KUKA KRL program: f1_Kuka_APT222T02S22.SRC

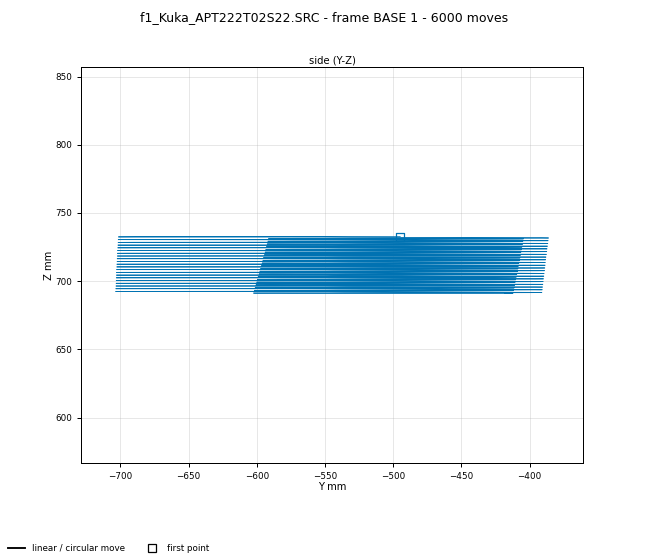
[picture p0: tool path of f1_Kuka_APT222T02S22.SRC in frame BASE 1, 6000 of 6001 moves have a stored position in this frame; points joined in program order, loops and branches not executed]
&ACCESS RVP
&REL 2
&PARAM TEMPLATE = C:\KRC\Roboter\Template\vorgabe
&PARAM EDITMASK = *
DEF f1_Kuka_APT222T02S22()


;FOLD INI;%{PE}%V3.2.0,%MKUKATPBASIS,%CINIT,%VCOMMON,%P
  ;FOLD BAS INI;%{E}%V3.2.0,%MKUKATPBASIS,%CINIT,%VINIT,%P
    GLOBAL INTERRUPT DECL 3 WHEN $STOPMESS==TRUE DO IR_STOPM ( )
    INTERRUPT ON 3
    BAS (#INITMOV,0 )
  ;ENDFOLD (BAS INI)
  ;FOLD USER INI;%{E}%V3.2.0,%MKUKATPUSER,%CINIT,%VINIT,%P
    ;Make your modifications here
  ;ENDFOLD (USER INI)
;ENDFOLD (INI)


;*** Make Null PTP Move
  PTP $pos_act

;*** Auto Load The Correct TOOL Data
  $tool=tool_data[2]

;*** Auto Load The Correct BASE Data
  $base=base_data[1]

  $ADVANCE = 5

;*** Restate Last Velocity
MMPM(30000.0)
SetRPM(8000)
LIN {X -0.072,Y -494.811,Z 732.685,A 0.000,B 0.000,C 90.000,E1 339.263} C_DIS
LIN {X 0.062,Y -499.458,Z 732.683,A 0.000,B 0.000,C 90.000,E1 338.847} C_DIS
LIN {X -0.040,Y -508.556,Z 732.679,A 0.000,B 0.000,C 90.000,E1 338.230} C_DIS
LIN {X -0.102,Y -530.986,Z 732.671,A 0.000,B 0.000,C 90.000,E1 336.847} C_DIS
LIN {X -0.056,Y -538.848,Z 732.669,A 0.000,B 0.000,C 90.000,E1 336.357} C_DIS
LIN {X 0.219,Y -546.203,Z 732.666,A 0.000,B 0.000,C 90.000,E1 335.793} C_DIS
LIN {X -0.007,Y -551.872,Z 732.663,A 0.000,B 0.000,C 90.000,E1 335.357} C_DIS
LIN {X 0.256,Y -559.941,Z 732.659,A 0.000,B 0.000,C 90.000,E1 334.588} C_DIS
LIN {X -0.047,Y -566.520,Z 732.655,A 0.000,B 0.000,C 90.000,E1 333.973} C_DIS
LIN {X -0.138,Y -575.282,Z 732.650,A 0.000,B 0.000,C 90.000,E1 333.050} C_DIS
LIN {X -0.034,Y -582.251,Z 732.646,A 0.000,B 0.000,C 90.000,E1 332.231} C_DIS
LIN {X -0.259,Y -591.121,Z 732.640,A 0.000,B 0.000,C 90.000,E1 331.179} C_DIS
LIN {X 0.245,Y -597.384,Z 732.635,A 0.000,B 0.000,C 90.000,E1 330.333} C_DIS
LIN {X 0.263,Y -604.345,Z 732.630,A 0.000,B 0.000,C 90.000,E1 329.410} C_DIS
LIN {X -0.134,Y -610.077,Z 732.626,A 0.000,B 0.000,C 90.000,E1 328.663} C_DIS
LIN {X 0.337,Y -617.212,Z 732.620,A 0.000,B 0.000,C 90.000,E1 327.582} C_DIS
LIN {X 0.048,Y -623.875,Z 732.614,A 0.000,B 0.000,C 90.000,E1 326.580} C_DIS
LIN {X 0.187,Y -628.508,Z 732.610,A 0.000,B 0.000,C 90.000,E1 325.801} C_DIS
LIN {X 0.019,Y -632.989,Z 732.606,A 0.000,B 0.000,C 90.000,E1 325.055} C_DIS
LIN {X -0.254,Y -637.926,Z 732.601,A 0.000,B 0.000,C 90.000,E1 324.196} C_DIS
LIN {X 0.036,Y -641.902,Z 732.597,A 0.000,B 0.000,C 90.000,E1 323.417} C_DIS
LIN {X -0.147,Y -645.788,Z 732.593,A 0.000,B 0.000,C 90.000,E1 322.683} C_DIS
LIN {X 0.221,Y -649.398,Z 732.589,A 0.000,B 0.000,C 90.000,E1 321.904} C_DIS
LIN {X 0.047,Y -653.994,Z 732.583,A 0.000,B 0.000,C 90.000,E1 320.928} C_DIS
LIN {X -0.062,Y -658.317,Z 732.578,A 0.000,B 0.000,C 90.000,E1 319.952} C_DIS
LIN {X 0.386,Y -662.353,Z 732.572,A 0.000,B 0.000,C 90.000,E1 318.933} C_DIS
LIN {X -0.109,Y -665.266,Z 732.568,A 0.000,B 0.000,C 90.000,E1 318.243} C_DIS
LIN {X 0.365,Y -667.979,Z 732.564,A 0.000,B 0.000,C 90.000,E1 317.472} C_DIS
LIN {X -0.061,Y -672.104,Z 732.557,A 0.000,B 0.000,C 90.000,E1 316.296} C_DIS
LIN {X 0.018,Y -675.195,Z 732.552,A 0.000,B 0.000,C 90.000,E1 315.324} C_DIS
LIN {X 0.141,Y -678.120,Z 732.547,A 0.000,B 0.000,C 90.000,E1 314.352} C_DIS
LIN {X -0.126,Y -681.503,Z 732.540,A 0.000,B 0.000,C 90.000,E1 313.176} C_DIS
LIN {X -0.340,Y -684.578,Z 732.533,A 0.000,B 0.000,C 90.000,E1 312.000} C_DIS
LIN {X 0.003,Y -687.418,Z 732.527,A 0.000,B 0.000,C 90.000,E1 310.782} C_DIS
LIN {X -0.202,Y -689.405,Z 732.521,A 0.000,B 0.000,C 90.000,E1 309.850} C_DIS
LIN {X -0.297,Y -691.088,Z 732.516,A 0.000,B 0.000,C 90.000,E1 308.910} C_DIS
LIN {X 0.064,Y -692.544,Z 732.511,A 0.000,B 0.000,C 90.000,E1 307.935} C_DIS
LIN {X 0.210,Y -694.120,Z 732.504,A 0.000,B 0.000,C 90.000,E1 306.744} C_DIS
LIN {X 0.181,Y -695.226,Z 732.499,A 0.000,B 0.000,C 90.000,E1 305.804} C_DIS
LIN {X -0.244,Y -696.182,Z 732.494,A 0.000,B 0.000,C 90.000,E1 304.898} C_DIS
LIN {X 0.204,Y -697.306,Z 732.486,A 0.000,B 0.000,C 90.000,E1 303.452} C_DIS
LIN {X -0.291,Y -698.505,Z 732.478,A 0.000,B 0.000,C 90.000,E1 302.084} C_DIS
LIN {X 0.163,Y -699.440,Z 732.472,A 0.000,B 0.000,C 90.000,E1 300.875} C_DIS
LIN {X 0.011,Y -699.898,Z 732.466,A 0.000,B 0.000,C 90.000,E1 299.951} C_DIS
LIN {X 0.137,Y -700.212,Z 732.460,A 0.000,B 0.000,C 90.000,E1 298.771} C_DIS
LIN {X -0.162,Y -700.761,Z 732.450,A 0.000,B 0.000,C 90.000,E1 296.924} C_DIS
LIN {X -0.116,Y -701.515,Z 732.440,A 0.000,B 0.000,C 90.000,E1 295.283} C_DIS
LIN {X -0.220,Y -701.426,Z 732.437,A 0.000,B 0.000,C 90.000,E1 294.591} C_DIS
LIN {X 0.329,Y -700.180,Z 732.434,A 0.000,B 0.000,C 90.000,E1 294.079} C_DIS
LIN {X -0.324,Y -699.415,Z 732.433,A 0.000,B 0.000,C 90.000,E1 293.898} C_DIS
LIN {X -0.190,Y -698.702,Z 732.432,A 0.000,B 0.000,C 90.000,E1 293.770} C_DIS
LIN {X 0.076,Y -696.517,Z 732.431,A 0.000,B 0.000,C 90.000,E1 293.515} C_DIS
LIN {X 0.347,Y -694.183,Z 732.429,A 0.000,B 0.000,C 90.000,E1 293.259} C_DIS
LIN {X 0.217,Y -692.875,Z 732.429,A 0.000,B 0.000,C 90.000,E1 293.153} C_DIS
LIN {X -0.223,Y -690.907,Z 732.428,A 0.000,B 0.000,C 90.000,E1 293.078} C_DIS
LIN {X -0.185,Y -686.403,Z 732.427,A 0.000,B 0.000,C 90.000,E1 292.898} C_DIS
LIN {X -0.121,Y -682.477,Z 732.427,A 0.000,B 0.000,C 90.000,E1 292.770} C_DIS
LIN {X 0.202,Y -676.428,Z 732.426,A 0.000,B 0.000,C 90.000,E1 292.589} C_DIS
LIN {X 0.149,Y -666.176,Z 732.425,A 0.000,B 0.000,C 90.000,E1 292.461} C_DIS
LIN {X 0.096,Y -652.560,Z 732.424,A 0.000,B 0.000,C 90.000,E1 292.280} C_DIS
LIN {X -0.358,Y -642.712,Z 732.423,A 0.000,B 0.000,C 90.000,E1 292.153} C_DIS
LIN {X 0.011,Y -629.339,Z 732.421,A 0.000,B 0.000,C 90.000,E1 291.844} C_DIS
LIN {X -0.078,Y -608.968,Z 732.419,A 0.000,B 0.000,C 90.000,E1 291.334} C_DIS
LIN {X -0.262,Y -581.079,Z 732.414,A 0.000,B 0.000,C 90.000,E1 290.556} C_DIS
LIN {X -0.251,Y -571.987,Z 732.413,A 0.000,B 0.000,C 90.000,E1 290.301} C_DIS
LIN {X 0.122,Y -566.747,Z 732.412,A 0.000,B 0.000,C 90.000,E1 290.120} C_DIS
LIN {X 0.007,Y -561.140,Z 732.411,A 0.000,B 0.000,C 90.000,E1 289.939} C_DIS
LIN {X -0.094,Y -556.625,Z 732.409,A 0.000,B 0.000,C 90.000,E1 289.685} C_DIS
LIN {X -0.122,Y -556.604,Z 732.409,A 0.000,B 0.000,C 90.000,E1 289.685} C_DIS
LIN {X -0.115,Y -555.581,Z 732.408,A 0.000,B 0.000,C 90.000,E1 289.504} C_DIS
LIN {X -0.129,Y -554.925,Z 732.406,A 0.000,B 0.000,C 90.000,E1 289.087} C_DIS
LIN {X 0.037,Y -554.116,Z 732.394,A 0.000,B 0.000,C 90.000,E1 286.913} C_DIS
LIN {X -0.146,Y -553.591,Z 732.386,A 0.000,B 0.000,C 90.000,E1 285.536} C_DIS
LIN {X -0.130,Y -552.835,Z 732.374,A 0.000,B 0.000,C 90.000,E1 283.300} C_DIS
LIN {X 0.286,Y -552.159,Z 732.363,A 0.000,B 0.000,C 90.000,E1 281.299} C_DIS
LIN {X 0.231,Y -551.598,Z 732.355,A 0.000,B 0.000,C 90.000,E1 279.905} C_DIS
LIN {X 0.170,Y -550.915,Z 732.347,A 0.000,B 0.000,C 90.000,E1 278.511} C_DIS
LIN {X 0.123,Y -550.135,Z 732.338,A 0.000,B 0.000,C 90.000,E1 276.834} C_DIS
LIN {X -0.008,Y -549.461,Z 732.329,A 0.000,B 0.000,C 90.000,E1 275.163} C_DIS
LIN {X 0.258,Y -549.002,Z 732.323,A 0.000,B 0.000,C 90.000,E1 274.012} C_DIS
LIN {X 0.072,Y -548.128,Z 732.312,A 0.000,B 0.000,C 90.000,E1 272.064} C_DIS
LIN {X -0.267,Y -547.557,Z 732.305,A 0.000,B 0.000,C 90.000,E1 270.974} C_DIS
LIN {X 0.009,Y -546.610,Z 732.296,A 0.000,B 0.000,C 90.000,E1 269.255} C_DIS
LIN {X 0.274,Y -545.503,Z 732.286,A 0.000,B 0.000,C 90.000,E1 267.535} C_DIS
LIN {X -0.068,Y -544.592,Z 732.279,A 0.000,B 0.000,C 90.000,E1 266.159} C_DIS
LIN {X 0.151,Y -543.656,Z 732.271,A 0.000,B 0.000,C 90.000,E1 264.723} C_DIS
LIN {X -0.122,Y -542.404,Z 732.261,A 0.000,B 0.000,C 90.000,E1 263.053} C_DIS
LIN {X 0.032,Y -541.731,Z 732.257,A 0.000,B 0.000,C 90.000,E1 262.186} C_DIS
LIN {X -0.058,Y -540.061,Z 732.246,A 0.000,B 0.000,C 90.000,E1 260.208} C_DIS
LIN {X -0.254,Y -538.600,Z 732.236,A 0.000,B 0.000,C 90.000,E1 258.522} C_DIS
LIN {X 0.077,Y -537.463,Z 732.228,A 0.000,B 0.000,C 90.000,E1 257.061} C_DIS
LIN {X -0.078,Y -536.456,Z 732.222,A 0.000,B 0.000,C 90.000,E1 255.936} C_DIS
LIN {X -0.002,Y -534.621,Z 732.212,A 0.000,B 0.000,C 90.000,E1 254.212} C_DIS
LIN {X 0.029,Y -532.802,Z 732.203,A 0.000,B 0.000,C 90.000,E1 252.489} C_DIS
LIN {X 0.146,Y -531.266,Z 732.195,A 0.000,B 0.000,C 90.000,E1 251.040} C_DIS
LIN {X 0.223,Y -529.733,Z 732.188,A 0.000,B 0.000,C 90.000,E1 249.880} C_DIS
LIN {X -0.032,Y -527.798,Z 732.180,A 0.000,B 0.000,C 90.000,E1 248.465} C_DIS
LIN {X -0.182,Y -526.562,Z 732.176,A 0.000,B 0.000,C 90.000,E1 247.614} C_DIS
LIN {X -0.298,Y -524.387,Z 732.168,A 0.000,B 0.000,C 90.000,E1 246.177} C_DIS
LIN {X 0.086,Y -522.509,Z 732.161,A 0.000,B 0.000,C 90.000,E1 244.973} C_DIS
LIN {X -0.024,Y -520.634,Z 732.155,A 0.000,B 0.000,C 90.000,E1 243.819} C_DIS
LIN {X -0.160,Y -518.571,Z 732.148,A 0.000,B 0.000,C 90.000,E1 242.666} C_DIS
LIN {X 0.144,Y -515.102,Z 732.138,A 0.000,B 0.000,C 90.000,E1 240.873} C_DIS
LIN {X -0.028,Y -512.842,Z 732.132,A 0.000,B 0.000,C 90.000,E1 239.715} C_DIS
LIN {X -0.138,Y -509.814,Z 732.124,A 0.000,B 0.000,C 90.000,E1 238.250} C_DIS
LIN {X 0.284,Y -506.094,Z 732.114,A 0.000,B 0.000,C 90.000,E1 236.421} C_DIS
LIN {X 0.104,Y -504.149,Z 732.109,A 0.000,B 0.000,C 90.000,E1 235.548} C_DIS
LIN {X -0.050,Y -500.700,Z 732.100,A 0.000,B 0.000,C 90.000,E1 234.069} C_DIS
LIN {X 0.159,Y -497.720,Z 732.094,A 0.000,B 0.000,C 90.000,E1 232.844} C_DIS
LIN {X 0.203,Y -492.397,Z 732.082,A 0.000,B 0.000,C 90.000,E1 230.723} C_DIS
LIN {X -0.125,Y -486.674,Z 732.068,A 0.000,B 0.000,C 90.000,E1 228.324} C_DIS
LIN {X 0.079,Y -482.573,Z 732.058,A 0.000,B 0.000,C 90.000,E1 226.458} C_DIS
LIN {X 0.174,Y -478.511,Z 732.048,A 0.000,B 0.000,C 90.000,E1 224.595} C_DIS
LIN {X 0.067,Y -475.211,Z 732.039,A 0.000,B 0.000,C 90.000,E1 223.056} C_DIS
LIN {X -0.083,Y -471.955,Z 732.031,A 0.000,B 0.000,C 90.000,E1 221.515} C_DIS
LIN {X -0.014,Y -469.158,Z 732.024,A 0.000,B 0.000,C 90.000,E1 220.253} C_DIS
LIN {X 0.020,Y -466.420,Z 732.017,A 0.000,B 0.000,C 90.000,E1 218.991} C_DIS
LIN {X -0.237,Y -462.911,Z 732.008,A 0.000,B 0.000,C 90.000,E1 217.443} C_DIS
LIN {X -0.089,Y -458.907,Z 731.997,A 0.000,B 0.000,C 90.000,E1 215.518} C_DIS
LIN {X 0.000,Y -453.311,Z 731.981,A 0.000,B 0.000,C 90.000,E1 212.625} C_DIS
LIN {X -0.135,Y -449.146,Z 731.969,A 0.000,B 0.000,C 90.000,E1 210.384} C_DIS
LIN {X -0.064,Y -444.919,Z 731.956,A 0.000,B 0.000,C 90.000,E1 208.103} C_DIS
LIN {X -0.199,Y -441.933,Z 731.947,A 0.000,B 0.000,C 90.000,E1 206.488} C_DIS
LIN {X 0.075,Y -437.662,Z 731.934,A 0.000,B 0.000,C 90.000,E1 204.155} C_DIS
LIN {X -0.004,Y -434.582,Z 731.925,A 0.000,B 0.000,C 90.000,E1 202.514} C_DIS
LIN {X -0.103,Y -430.855,Z 731.914,A 0.000,B 0.000,C 90.000,E1 200.536} C_DIS
LIN {X -0.195,Y -428.421,Z 731.907,A 0.000,B 0.000,C 90.000,E1 199.214} C_DIS
LIN {X 0.015,Y -425.318,Z 731.897,A 0.000,B 0.000,C 90.000,E1 197.511} C_DIS
LIN {X 0.082,Y -421.438,Z 731.886,A 0.000,B 0.000,C 90.000,E1 195.481} C_DIS
LIN {X -0.003,Y -417.151,Z 731.873,A 0.000,B 0.000,C 90.000,E1 193.119} C_DIS
LIN {X -0.064,Y -414.186,Z 731.863,A 0.000,B 0.000,C 90.000,E1 191.422} C_DIS
LIN {X -0.095,Y -409.393,Z 731.848,A 0.000,B 0.000,C 90.000,E1 188.681} C_DIS
LIN {X -0.082,Y -406.083,Z 731.837,A 0.000,B 0.000,C 90.000,E1 186.606} C_DIS
LIN {X -0.138,Y -403.460,Z 731.827,A 0.000,B 0.000,C 90.000,E1 184.878} C_DIS
LIN {X -0.075,Y -398.689,Z 731.808,A 0.000,B 0.000,C 90.000,E1 181.375} C_DIS
LIN {X 0.111,Y -397.027,Z 731.800,A 0.000,B 0.000,C 90.000,E1 179.943} C_DIS
LIN {X 0.154,Y -394.849,Z 731.788,A 0.000,B 0.000,C 90.000,E1 177.822} C_DIS
LIN {X -0.105,Y -393.435,Z 731.780,A 0.000,B 0.000,C 90.000,E1 176.445} C_DIS
LIN {X 0.140,Y -391.072,Z 731.764,A 0.000,B 0.000,C 90.000,E1 173.571} C_DIS
LIN {X -0.112,Y -388.928,Z 731.743,A 0.000,B 0.000,C 90.000,E1 169.690} C_DIS
LIN {X 0.108,Y -388.364,Z 731.735,A 0.000,B 0.000,C 90.000,E1 168.229} C_DIS
LIN {X -0.107,Y -387.578,Z 731.723,A 0.000,B 0.000,C 90.000,E1 166.117} C_DIS
LIN {X -0.178,Y -387.074,Z 731.713,A 0.000,B 0.000,C 90.000,E1 164.338} C_DIS
LIN {X -0.097,Y -386.682,Z 731.699,A 0.000,B 0.000,C 90.000,E1 161.819} C_DIS
LIN {X 0.061,Y -386.356,Z 731.687,A 0.000,B 0.000,C 90.000,E1 159.645} C_DIS
LIN {X 0.113,Y -386.156,Z 731.675,A 0.000,B 0.000,C 90.000,E1 157.486} C_DIS
LIN {X -0.213,Y -386.059,Z 731.659,A 0.000,B 0.000,C 90.000,E1 154.665} C_DIS
LIN {X 0.138,Y -386.635,Z 731.641,A 0.000,B 0.000,C 90.000,E1 151.385} C_DIS
LIN {X 0.086,Y -388.356,Z 731.619,A 0.000,B 0.000,C 90.000,E1 147.454} C_DIS
LIN {X 0.203,Y -389.389,Z 731.611,A 0.000,B 0.000,C 90.000,E1 146.008} C_DIS
LIN {X -0.150,Y -392.284,Z 731.596,A 0.000,B 0.000,C 90.000,E1 143.210} C_DIS
LIN {X 0.022,Y -394.681,Z 731.586,A 0.000,B 0.000,C 90.000,E1 141.412} C_DIS
LIN {X -0.105,Y -395.679,Z 731.582,A 0.000,B 0.000,C 90.000,E1 140.723} C_DIS
LIN {X -0.120,Y -397.732,Z 731.576,A 0.000,B 0.000,C 90.000,E1 139.666} C_DIS
LIN {X 0.085,Y -399.513,Z 731.572,A 0.000,B 0.000,C 90.000,E1 138.933} C_DIS
LIN {X 0.096,Y -401.109,Z 731.569,A 0.000,B 0.000,C 90.000,E1 138.405} C_DIS
LIN {X 0.011,Y -403.546,Z 731.566,A 0.000,B 0.000,C 90.000,E1 137.838} C_DIS
LIN {X -0.075,Y -406.596,Z 731.563,A 0.000,B 0.000,C 90.000,E1 137.310} C_DIS
LIN {X 0.042,Y -410.568,Z 731.560,A 0.000,B 0.000,C 90.000,E1 136.743} C_DIS
LIN {X -0.164,Y -416.992,Z 731.556,A 0.000,B 0.000,C 90.000,E1 136.053} C_DIS
LIN {X -0.115,Y -439.152,Z 731.544,A 0.000,B 0.000,C 90.000,E1 133.866} C_DIS
LIN {X -0.267,Y -450.970,Z 731.537,A 0.000,B 0.000,C 90.000,E1 132.771} C_DIS
LIN {X 0.144,Y -456.781,Z 731.534,A 0.000,B 0.000,C 90.000,E1 132.162} C_DIS
LIN {X -0.188,Y -465.234,Z 731.530,A 0.000,B 0.000,C 90.000,E1 131.391} C_DIS
LIN {X 0.117,Y -474.954,Z 731.524,A 0.000,B 0.000,C 90.000,E1 130.378} C_DIS
LIN {X -0.015,Y -480.291,Z 731.521,A 0.000,B 0.000,C 90.000,E1 129.850} C_DIS
LIN {X -0.139,Y -488.498,Z 731.517,A 0.000,B 0.000,C 90.000,E1 128.991} C_DIS
LIN {X -0.288,Y -493.488,Z 731.514,A 0.000,B 0.000,C 90.000,E1 128.463} C_DIS
LIN {X -0.219,Y -498.354,Z 731.510,A 0.000,B 0.000,C 90.000,E1 127.890} C_DIS
LIN {X 0.225,Y -503.166,Z 731.507,A 0.000,B 0.000,C 90.000,E1 127.237} C_DIS
LIN {X 0.005,Y -510.954,Z 731.501,A 0.000,B 0.000,C 90.000,E1 126.217} C_DIS
LIN {X 0.250,Y -515.011,Z 731.498,A 0.000,B 0.000,C 90.000,E1 125.598} C_DIS
LIN {X 0.046,Y -520.356,Z 731.493,A 0.000,B 0.000,C 90.000,E1 124.739} C_DIS
LIN {X -0.188,Y -522.943,Z 731.491,A 0.000,B 0.000,C 90.000,E1 124.326} C_DIS
LIN {X 0.116,Y -527.468,Z 731.486,A 0.000,B 0.000,C 90.000,E1 123.420} C_DIS
LIN {X 0.053,Y -530.992,Z 731.482,A 0.000,B 0.000,C 90.000,E1 122.704} C_DIS
LIN {X -0.139,Y -534.239,Z 731.478,A 0.000,B 0.000,C 90.000,E1 122.005} C_DIS
LIN {X -0.004,Y -539.110,Z 731.471,A 0.000,B 0.000,C 90.000,E1 120.846} C_DIS
LIN {X -0.084,Y -543.694,Z 731.465,A 0.000,B 0.000,C 90.000,E1 119.716} C_DIS
LIN {X -0.118,Y -546.991,Z 731.460,A 0.000,B 0.000,C 90.000,E1 118.871} C_DIS
LIN {X 0.134,Y -551.138,Z 731.454,A 0.000,B 0.000,C 90.000,E1 117.719} C_DIS
LIN {X -0.039,Y -554.859,Z 731.448,A 0.000,B 0.000,C 90.000,E1 116.616} C_DIS
LIN {X 0.045,Y -557.308,Z 731.443,A 0.000,B 0.000,C 90.000,E1 115.771} C_DIS
LIN {X -0.090,Y -559.424,Z 731.439,A 0.000,B 0.000,C 90.000,E1 114.951} C_DIS
LIN {X 0.309,Y -561.306,Z 731.434,A 0.000,B 0.000,C 90.000,E1 114.079} C_DIS
LIN {X 0.218,Y -562.944,Z 731.429,A 0.000,B 0.000,C 90.000,E1 113.259} C_DIS
LIN {X 0.247,Y -564.707,Z 731.423,A 0.000,B 0.000,C 90.000,E1 112.153} C_DIS
LIN {X -0.084,Y -567.242,Z 731.414,A 0.000,B 0.000,C 90.000,E1 110.536} C_DIS
LIN {X -0.191,Y -568.889,Z 731.408,A 0.000,B 0.000,C 90.000,E1 109.450} C_DIS
LIN {X -0.299,Y -571.141,Z 731.399,A 0.000,B 0.000,C 90.000,E1 107.819} C_DIS
LIN {X 0.180,Y -573.194,Z 731.390,A 0.000,B 0.000,C 90.000,E1 106.134} C_DIS
LIN {X 0.189,Y -574.869,Z 731.382,A 0.000,B 0.000,C 90.000,E1 104.773} C_DIS
LIN {X 0.229,Y -576.550,Z 731.375,A 0.000,B 0.000,C 90.000,E1 103.411} C_DIS
LIN {X -0.186,Y -578.528,Z 731.366,A 0.000,B 0.000,C 90.000,E1 101.827} C_DIS
LIN {X -0.104,Y -580.501,Z 731.357,A 0.000,B 0.000,C 90.000,E1 100.197} C_DIS
LIN {X 0.138,Y -581.751,Z 731.351,A 0.000,B 0.000,C 90.000,E1 99.095} C_DIS
LIN {X 0.052,Y -583.153,Z 731.343,A 0.000,B 0.000,C 90.000,E1 97.757} C_DIS
LIN {X 0.066,Y -584.719,Z 731.334,A 0.000,B 0.000,C 90.000,E1 96.144} C_DIS
LIN {X 0.114,Y -586.280,Z 731.325,A 0.000,B 0.000,C 90.000,E1 94.531} C_DIS
LIN {X 0.138,Y -587.665,Z 731.316,A 0.000,B 0.000,C 90.000,E1 92.922} C_DIS
LIN {X -0.256,Y -588.499,Z 731.310,A 0.000,B 0.000,C 90.000,E1 91.892} C_DIS
LIN {X -0.215,Y -589.463,Z 731.302,A 0.000,B 0.000,C 90.000,E1 90.286} C_DIS
LIN {X 0.216,Y -590.160,Z 731.294,A 0.000,B 0.000,C 90.000,E1 88.912} C_DIS
LIN {X 0.287,Y -590.716,Z 731.285,A 0.000,B 0.000,C 90.000,E1 87.306} C_DIS
LIN {X -0.044,Y -590.996,Z 731.279,A 0.000,B 0.000,C 90.000,E1 86.274} C_DIS
LIN {X -0.125,Y -591.225,Z 731.272,A 0.000,B 0.000,C 90.000,E1 84.951} C_DIS
LIN {X 0.190,Y -591.332,Z 731.266,A 0.000,B 0.000,C 90.000,E1 83.856} C_DIS
LIN {X -0.217,Y -591.373,Z 731.257,A 0.000,B 0.000,C 90.000,E1 82.299} C_DIS
LIN {X 0.175,Y -591.261,Z 731.251,A 0.000,B 0.000,C 90.000,E1 81.197} C_DIS
LIN {X 0.254,Y -590.970,Z 731.244,A 0.000,B 0.000,C 90.000,E1 79.859} C_DIS
LIN {X -0.257,Y -590.376,Z 731.236,A 0.000,B 0.000,C 90.000,E1 78.578} C_DIS
LIN {X 0.181,Y -589.551,Z 731.228,A 0.000,B 0.000,C 90.000,E1 76.937} C_DIS
LIN {X 0.014,Y -588.573,Z 731.219,A 0.000,B 0.000,C 90.000,E1 75.353} C_DIS
LIN {X -0.125,Y -587.614,Z 731.211,A 0.000,B 0.000,C 90.000,E1 74.031} C_DIS
LIN {X -0.112,Y -586.791,Z 731.205,A 0.000,B 0.000,C 90.000,E1 72.960} C_DIS
LIN {X 0.061,Y -585.887,Z 731.199,A 0.000,B 0.000,C 90.000,E1 71.873} C_DIS
LIN {X 0.296,Y -584.334,Z 731.190,A 0.000,B 0.000,C 90.000,E1 70.242} C_DIS
LIN {X 0.224,Y -583.512,Z 731.186,A 0.000,B 0.000,C 90.000,E1 69.444} C_DIS
LIN {X 0.195,Y -581.944,Z 731.179,A 0.000,B 0.000,C 90.000,E1 68.103} C_DIS
LIN {X -0.047,Y -580.554,Z 731.173,A 0.000,B 0.000,C 90.000,E1 67.050} C_DIS
LIN {X -0.077,Y -578.972,Z 731.167,A 0.000,B 0.000,C 90.000,E1 65.973} C_DIS
LIN {X 0.258,Y -576.731,Z 731.159,A 0.000,B 0.000,C 90.000,E1 64.588} C_DIS
LIN {X -0.186,Y -575.191,Z 731.154,A 0.000,B 0.000,C 90.000,E1 63.819} C_DIS
LIN {X 0.060,Y -572.304,Z 731.147,A 0.000,B 0.000,C 90.000,E1 62.436} C_DIS
LIN {X -0.165,Y -570.297,Z 731.142,A 0.000,B 0.000,C 90.000,E1 61.641} C_DIS
LIN {X 0.094,Y -568.119,Z 731.138,A 0.000,B 0.000,C 90.000,E1 60.795} C_DIS
LIN {X -0.067,Y -564.923,Z 731.132,A 0.000,B 0.000,C 90.000,E1 59.715} C_DIS
LIN {X -0.072,Y -561.323,Z 731.126,A 0.000,B 0.000,C 90.000,E1 58.614} C_DIS
LIN {X -0.192,Y -559.412,Z 731.123,A 0.000,B 0.000,C 90.000,E1 58.074} C_DIS
LIN {X -0.025,Y -557.376,Z 731.120,A 0.000,B 0.000,C 90.000,E1 57.502} C_DIS
LIN {X 0.371,Y -553.929,Z 731.115,A 0.000,B 0.000,C 90.000,E1 56.628} C_DIS
LIN {X 0.256,Y -550.048,Z 731.110,A 0.000,B 0.000,C 90.000,E1 55.801} C_DIS
LIN {X 0.053,Y -547.302,Z 731.107,A 0.000,B 0.000,C 90.000,E1 55.261} C_DIS
LIN {X 0.177,Y -542.592,Z 731.102,A 0.000,B 0.000,C 90.000,E1 54.402} C_DIS
LIN {X -0.084,Y -539.262,Z 731.099,A 0.000,B 0.000,C 90.000,E1 53.863} C_DIS
LIN {X 0.114,Y -536.663,Z 731.097,A 0.000,B 0.000,C 90.000,E1 53.417} C_DIS
LIN {X -0.166,Y -531.914,Z 731.093,A 0.000,B 0.000,C 90.000,E1 52.763} C_DIS
LIN {X -0.003,Y -528.732,Z 731.091,A 0.000,B 0.000,C 90.000,E1 52.316} C_DIS
LIN {X 0.235,Y -523.054,Z 731.087,A 0.000,B 0.000,C 90.000,E1 51.618} C_DIS
LIN {X -0.041,Y -519.061,Z 731.085,A 0.000,B 0.000,C 90.000,E1 51.215} C_DIS
LIN {X -0.029,Y -514.796,Z 731.082,A 0.000,B 0.000,C 90.000,E1 50.803} C_DIS
LIN {X 0.055,Y -508.854,Z 731.079,A 0.000,B 0.000,C 90.000,E1 50.275} C_DIS
LIN {X -0.020,Y -504.293,Z 731.077,A 0.000,B 0.000,C 90.000,E1 49.908} C_DIS
LIN {X -0.206,Y -497.897,Z 731.075,A 0.000,B 0.000,C 90.000,E1 49.461} C_DIS
LIN {X 0.090,Y -493.065,Z 731.073,A 0.000,B 0.000,C 90.000,E1 49.094} C_DIS
LIN {X -0.068,Y -485.326,Z 731.070,A 0.000,B 0.000,C 90.000,E1 48.609} C_DIS
LIN {X -0.089,Y -472.141,Z 731.066,A 0.000,B 0.000,C 90.000,E1 47.796} C_DIS
LIN {X 0.098,Y -454.360,Z 731.059,A 0.000,B 0.000,C 90.000,E1 46.662} C_DIS
LIN {X -0.155,Y -428.756,Z 731.050,A 0.000,B 0.000,C 90.000,E1 45.000} C_DIS
LIN {X 0.160,Y -422.659,Z 731.047,A 0.000,B 0.000,C 90.000,E1 44.514} C_DIS
LIN {X -0.258,Y -416.837,Z 731.045,A 0.000,B 0.000,C 90.000,E1 44.109} C_DIS
LIN {X 0.003,Y -416.824,Z 731.045,A 0.000,B 0.000,C 90.000,E1 44.069} C_DIS
LIN {X 0.116,Y -407.449,Z 731.019,A 0.000,B 0.000,C 90.000,E1 39.439} C_DIS
LIN {X 0.241,Y -405.716,Z 731.013,A 0.000,B 0.000,C 90.000,E1 38.382} C_DIS
LIN {X 0.042,Y -404.547,Z 731.011,A 0.000,B 0.000,C 90.000,E1 37.890} C_DIS
LIN {X -0.007,Y -405.117,Z 730.990,A 0.000,B 0.000,C 90.000,E1 34.246} C_DIS
LIN {X 0.105,Y -406.070,Z 730.977,A 0.000,B 0.000,C 90.000,E1 31.799} C_DIS
LIN {X -0.173,Y -407.225,Z 730.963,A 0.000,B 0.000,C 90.000,E1 29.411} C_DIS
LIN {X 0.015,Y -408.387,Z 730.952,A 0.000,B 0.000,C 90.000,E1 27.308} C_DIS
LIN {X -0.050,Y -409.945,Z 730.938,A 0.000,B 0.000,C 90.000,E1 24.899} C_DIS
LIN {X 0.144,Y -411.908,Z 730.925,A 0.000,B 0.000,C 90.000,E1 22.461} C_DIS
LIN {X -0.193,Y -413.507,Z 730.915,A 0.000,B 0.000,C 90.000,E1 20.791} C_DIS
LIN {X -0.113,Y -415.694,Z 730.904,A 0.000,B 0.000,C 90.000,E1 18.725} C_DIS
LIN {X 0.047,Y -418.653,Z 730.891,A 0.000,B 0.000,C 90.000,E1 16.315} C_DIS
LIN {X 0.051,Y -421.924,Z 730.878,A 0.000,B 0.000,C 90.000,E1 13.939} C_DIS
LIN {X -0.232,Y -424.858,Z 730.866,A 0.000,B 0.000,C 90.000,E1 11.951} C_DIS
LIN {X 0.080,Y -428.405,Z 730.853,A 0.000,B 0.000,C 90.000,E1 9.557} C_DIS
LIN {X -0.191,Y -431.434,Z 730.842,A 0.000,B 0.000,C 90.000,E1 7.587} C_DIS
LIN {X 0.186,Y -435.515,Z 730.827,A 0.000,B 0.000,C 90.000,E1 4.878} C_DIS
LIN {X -0.024,Y -438.842,Z 730.816,A 0.000,B 0.000,C 90.000,E1 2.922} C_DIS
LIN {X -0.087,Y -442.964,Z 730.803,A 0.000,B 0.000,C 90.000,E1 0.630} C_DIS
LIN {X -0.177,Y -447.066,Z 730.792,A 0.000,B 0.000,C 90.000,E1 358.511} C_DIS
LIN {X -0.100,Y -452.999,Z 730.775,A 0.000,B 0.000,C 90.000,E1 355.584} C_DIS
LIN {X 0.105,Y -457.219,Z 730.765,A 0.000,B 0.000,C 90.000,E1 353.628} C_DIS
LIN {X -0.175,Y -460.629,Z 730.756,A 0.000,B 0.000,C 90.000,E1 352.064} C_DIS
LIN {X 0.070,Y -463.938,Z 730.747,A 0.000,B 0.000,C 90.000,E1 350.443} C_DIS
LIN {X 0.190,Y -466.495,Z 730.740,A 0.000,B 0.000,C 90.000,E1 349.162} C_DIS
LIN {X -0.112,Y -468.882,Z 730.733,A 0.000,B 0.000,C 90.000,E1 347.937} C_DIS
LIN {X -0.004,Y -471.755,Z 730.724,A 0.000,B 0.000,C 90.000,E1 346.353} C_DIS
LIN {X -0.186,Y -474.593,Z 730.716,A 0.000,B 0.000,C 90.000,E1 344.810} C_DIS
LIN {X -0.078,Y -479.484,Z 730.702,A 0.000,B 0.000,C 90.000,E1 342.308} C_DIS
LIN {X -0.272,Y -481.829,Z 730.697,A 0.000,B 0.000,C 90.000,E1 341.402} C_DIS
LIN {X 0.173,Y -483.778,Z 730.693,A 0.000,B 0.000,C 90.000,E1 340.732} C_DIS
LIN {X -0.140,Y -486.177,Z 730.690,A 0.000,B 0.000,C 90.000,E1 340.242} C_DIS
LIN {X -0.127,Y -487.850,Z 730.688,A 0.000,B 0.000,C 90.000,E1 339.934} C_DIS
LIN {X 0.136,Y -491.112,Z 730.686,A 0.000,B 0.000,C 90.000,E1 339.444} C_DIS
LIN {X -0.104,Y -495.262,Z 730.683,A 0.000,B 0.000,C 90.000,E1 339.028} C_DIS
LIN {X -0.112,Y -502.208,Z 730.680,A 0.000,B 0.000,C 90.000,E1 338.465} C_DIS
LIN {X 0.212,Y -522.720,Z 730.673,A 0.000,B 0.000,C 90.000,E1 337.102} C_DIS
LIN {X -0.022,Y -535.363,Z 730.669,A 0.000,B 0.000,C 90.000,E1 336.357} C_DIS
LIN {X 0.055,Y -539.919,Z 730.667,A 0.000,B 0.000,C 90.000,E1 336.049} C_DIS
LIN {X 0.214,Y -547.288,Z 730.664,A 0.000,B 0.000,C 90.000,E1 335.485} C_DIS
LIN {X 0.088,Y -551.503,Z 730.662,A 0.000,B 0.000,C 90.000,E1 335.153} C_DIS
LIN {X 0.081,Y -559.673,Z 730.658,A 0.000,B 0.000,C 90.000,E1 334.409} C_DIS
LIN {X 0.064,Y -566.233,Z 730.654,A 0.000,B 0.000,C 90.000,E1 333.768} C_DIS
LIN {X -0.215,Y -573.776,Z 730.650,A 0.000,B 0.000,C 90.000,E1 332.999} C_DIS
LIN {X 0.165,Y -580.860,Z 730.645,A 0.000,B 0.000,C 90.000,E1 332.153} C_DIS
LIN {X 0.089,Y -585.299,Z 730.643,A 0.000,B 0.000,C 90.000,E1 331.641} C_DIS
LIN {X 0.016,Y -591.901,Z 730.638,A 0.000,B 0.000,C 90.000,E1 330.845} C_DIS
LIN {X -0.029,Y -599.178,Z 730.633,A 0.000,B 0.000,C 90.000,E1 329.921} C_DIS
LIN {X 0.009,Y -606.107,Z 730.628,A 0.000,B 0.000,C 90.000,E1 328.997} C_DIS
LIN {X 0.151,Y -611.763,Z 730.623,A 0.000,B 0.000,C 90.000,E1 328.201} C_DIS
LIN {X -0.173,Y -617.098,Z 730.619,A 0.000,B 0.000,C 90.000,E1 327.454} C_DIS
LIN {X -0.118,Y -622.985,Z 730.614,A 0.000,B 0.000,C 90.000,E1 326.548} C_DIS
LIN {X 0.189,Y -626.908,Z 730.611,A 0.000,B 0.000,C 90.000,E1 325.881} C_DIS
LIN {X 0.004,Y -631.496,Z 730.606,A 0.000,B 0.000,C 90.000,E1 325.135} C_DIS
LIN {X -0.262,Y -636.534,Z 730.601,A 0.000,B 0.000,C 90.000,E1 324.276} C_DIS
LIN {X -0.103,Y -641.896,Z 730.596,A 0.000,B 0.000,C 90.000,E1 323.256} C_DIS
LIN {X 0.230,Y -645.766,Z 730.592,A 0.000,B 0.000,C 90.000,E1 322.477} C_DIS
LIN {X -0.327,Y -648.814,Z 730.588,A 0.000,B 0.000,C 90.000,E1 321.904} C_DIS
LIN {X -0.004,Y -653.482,Z 730.583,A 0.000,B 0.000,C 90.000,E1 320.884} C_DIS
LIN {X -0.127,Y -657.901,Z 730.577,A 0.000,B 0.000,C 90.000,E1 319.908} C_DIS
LIN {X -0.217,Y -662.975,Z 730.570,A 0.000,B 0.000,C 90.000,E1 318.690} C_DIS
LIN {X -0.222,Y -666.803,Z 730.565,A 0.000,B 0.000,C 90.000,E1 317.715} C_DIS
LIN {X 0.278,Y -671.038,Z 730.558,A 0.000,B 0.000,C 90.000,E1 316.458} C_DIS
LIN {X 0.368,Y -675.015,Z 730.552,A 0.000,B 0.000,C 90.000,E1 315.243} C_DIS
LIN {X 0.004,Y -677.969,Z 730.546,A 0.000,B 0.000,C 90.000,E1 314.312} C_DIS
LIN {X 0.222,Y -681.397,Z 730.540,A 0.000,B 0.000,C 90.000,E1 313.095} C_DIS
LIN {X 0.007,Y -684.528,Z 730.533,A 0.000,B 0.000,C 90.000,E1 311.919} C_DIS
LIN {X 0.350,Y -687.381,Z 730.526,A 0.000,B 0.000,C 90.000,E1 310.701} C_DIS
LIN {X 0.083,Y -688.951,Z 730.522,A 0.000,B 0.000,C 90.000,E1 310.011} C_DIS
LIN {X -0.015,Y -690.741,Z 730.517,A 0.000,B 0.000,C 90.000,E1 309.072} C_DIS
LIN {X 0.347,Y -692.289,Z 730.512,A 0.000,B 0.000,C 90.000,E1 308.096} C_DIS
LIN {X 0.296,Y -693.603,Z 730.507,A 0.000,B 0.000,C 90.000,E1 307.156} C_DIS
LIN {X -0.094,Y -695.094,Z 730.500,A 0.000,B 0.000,C 90.000,E1 306.011} C_DIS
LIN {X 0.100,Y -696.307,Z 730.494,A 0.000,B 0.000,C 90.000,E1 304.818} C_DIS
LIN {X -0.037,Y -697.451,Z 730.486,A 0.000,B 0.000,C 90.000,E1 303.420} C_DIS
LIN {X 0.049,Y -698.648,Z 730.478,A 0.000,B 0.000,C 90.000,E1 302.005} C_DIS
LIN {X -0.100,Y -699.588,Z 730.471,A 0.000,B 0.000,C 90.000,E1 300.846} C_DIS
LIN {X 0.082,Y -699.952,Z 730.467,A 0.000,B 0.000,C 90.000,E1 300.129} C_DIS
LIN {X -0.144,Y -700.334,Z 730.460,A 0.000,B 0.000,C 90.000,E1 298.743} C_DIS
LIN {X -0.077,Y -700.730,Z 730.452,A 0.000,B 0.000,C 90.000,E1 297.334} C_DIS
LIN {X -0.071,Y -701.533,Z 730.441,A 0.000,B 0.000,C 90.000,E1 295.463} C_DIS
LIN {X 0.204,Y -701.653,Z 730.440,A 0.000,B 0.000,C 90.000,E1 295.207} C_DIS
LIN {X -0.177,Y -701.589,Z 730.438,A 0.000,B 0.000,C 90.000,E1 294.771} C_DIS
LIN {X 0.098,Y -701.433,Z 730.436,A 0.000,B 0.000,C 90.000,E1 294.515} C_DIS
LIN {X -0.282,Y -700.101,Z 730.434,A 0.000,B 0.000,C 90.000,E1 294.079} C_DIS
LIN {X -0.012,Y -699.181,Z 730.432,A 0.000,B 0.000,C 90.000,E1 293.823} C_DIS
LIN {X 0.122,Y -698.335,Z 730.432,A 0.000,B 0.000,C 90.000,E1 293.695} C_DIS
LIN {X 0.237,Y -694.817,Z 730.430,A 0.000,B 0.000,C 90.000,E1 293.334} C_DIS
LIN {X -0.267,Y -693.464,Z 730.429,A 0.000,B 0.000,C 90.000,E1 293.259} C_DIS
LIN {X -0.132,Y -691.841,Z 730.428,A 0.000,B 0.000,C 90.000,E1 293.131} C_DIS
LIN {X -0.068,Y -689.586,Z 730.428,A 0.000,B 0.000,C 90.000,E1 293.025} C_DIS
LIN {X 0.121,Y -685.177,Z 730.427,A 0.000,B 0.000,C 90.000,E1 292.845} C_DIS
LIN {X 0.075,Y -677.437,Z 730.426,A 0.000,B 0.000,C 90.000,E1 292.642} C_DIS
LIN {X -0.205,Y -672.281,Z 730.425,A 0.000,B 0.000,C 90.000,E1 292.589} C_DIS
LIN {X 0.217,Y -655.341,Z 730.424,A 0.000,B 0.000,C 90.000,E1 292.333} C_DIS
LIN {X -0.165,Y -645.429,Z 730.423,A 0.000,B 0.000,C 90.000,E1 292.206} C_DIS
LIN {X 0.307,Y -632.078,Z 730.422,A 0.000,B 0.000,C 90.000,E1 291.897} C_DIS
LIN {X -0.241,Y -622.305,Z 730.421,A 0.000,B 0.000,C 90.000,E1 291.716} C_DIS
LIN {X -0.141,Y -601.467,Z 730.417,A 0.000,B 0.000,C 90.000,E1 291.153} C_DIS
LIN {X -0.258,Y -580.473,Z 730.414,A 0.000,B 0.000,C 90.000,E1 290.556} C_DIS
LIN {X -0.245,Y -571.361,Z 730.413,A 0.000,B 0.000,C 90.000,E1 290.301} C_DIS
LIN {X 0.061,Y -567.693,Z 730.412,A 0.000,B 0.000,C 90.000,E1 290.174} C_DIS
LIN {X 0.150,Y -561.118,Z 730.411,A 0.000,B 0.000,C 90.000,E1 289.939} C_DIS
LIN {X 0.092,Y -556.671,Z 730.409,A 0.000,B 0.000,C 90.000,E1 289.685} C_DIS
LIN {X 0.063,Y -556.626,Z 730.409,A 0.000,B 0.000,C 90.000,E1 289.685} C_DIS
LIN {X -0.074,Y -555.554,Z 730.408,A 0.000,B 0.000,C 90.000,E1 289.504} C_DIS
LIN {X -0.086,Y -554.899,Z 730.406,A 0.000,B 0.000,C 90.000,E1 289.087} C_DIS
LIN {X 0.221,Y -554.301,Z 730.397,A 0.000,B 0.000,C 90.000,E1 287.457} C_DIS
LIN {X 0.162,Y -553.684,Z 730.388,A 0.000,B 0.000,C 90.000,E1 285.788} C_DIS
LIN {X -0.091,Y -552.807,Z 730.374,A 0.000,B 0.000,C 90.000,E1 283.300} C_DIS
LIN {X 0.208,Y -552.247,Z 730.365,A 0.000,B 0.000,C 90.000,E1 281.591} C_DIS
LIN {X 0.154,Y -551.691,Z 730.357,A 0.000,B 0.000,C 90.000,E1 280.197} C_DIS
LIN {X 0.097,Y -551.043,Z 730.349,A 0.000,B 0.000,C 90.000,E1 278.803} C_DIS
LIN {X 0.161,Y -550.106,Z 730.338,A 0.000,B 0.000,C 90.000,E1 276.834} C_DIS
LIN {X -0.064,Y -549.560,Z 730.330,A 0.000,B 0.000,C 90.000,E1 275.454} C_DIS
LIN {X 0.211,Y -549.161,Z 730.324,A 0.000,B 0.000,C 90.000,E1 274.302} C_DIS
LIN {X 0.014,Y -548.386,Z 730.315,A 0.000,B 0.000,C 90.000,E1 272.636} C_DIS
LIN {X 0.224,Y -547.905,Z 730.308,A 0.000,B 0.000,C 90.000,E1 271.489} C_DIS
LIN {X -0.087,Y -547.148,Z 730.301,A 0.000,B 0.000,C 90.000,E1 270.115} C_DIS
LIN {X 0.093,Y -546.454,Z 730.294,A 0.000,B 0.000,C 90.000,E1 268.969} C_DIS
LIN {X -0.192,Y -545.379,Z 730.285,A 0.000,B 0.000,C 90.000,E1 267.306} C_DIS
LIN {X 0.043,Y -544.462,Z 730.277,A 0.000,B 0.000,C 90.000,E1 265.869} C_DIS
LIN {X 0.267,Y -543.489,Z 730.269,A 0.000,B 0.000,C 90.000,E1 264.432} C_DIS
LIN {X -0.003,Y -542.250,Z 730.260,A 0.000,B 0.000,C 90.000,E1 262.761} C_DIS
LIN {X -0.163,Y -540.567,Z 730.249,A 0.000,B 0.000,C 90.000,E1 260.792} C_DIS
LIN {X 0.110,Y -539.345,Z 730.241,A 0.000,B 0.000,C 90.000,E1 259.342} C_DIS
LIN {X 0.059,Y -537.736,Z 730.230,A 0.000,B 0.000,C 90.000,E1 257.353} C_DIS
LIN {X -0.033,Y -536.461,Z 730.222,A 0.000,B 0.000,C 90.000,E1 255.936} C_DIS
LIN {X -0.147,Y -534.964,Z 730.214,A 0.000,B 0.000,C 90.000,E1 254.519} C_DIS
LIN {X 0.043,Y -533.135,Z 730.204,A 0.000,B 0.000,C 90.000,E1 252.779} C_DIS
LIN {X 0.192,Y -531.328,Z 730.195,A 0.000,B 0.000,C 90.000,E1 251.040} C_DIS
LIN {X 0.271,Y -529.795,Z 730.188,A 0.000,B 0.000,C 90.000,E1 249.880} C_DIS
LIN {X 0.018,Y -527.860,Z 730.180,A 0.000,B 0.000,C 90.000,E1 248.465} C_DIS
LIN {X 0.040,Y -526.171,Z 730.174,A 0.000,B 0.000,C 90.000,E1 247.305} C_DIS
LIN {X -0.247,Y -524.453,Z 730.168,A 0.000,B 0.000,C 90.000,E1 246.177} C_DIS
LIN {X 0.137,Y -522.571,Z 730.161,A 0.000,B 0.000,C 90.000,E1 244.973} C_DIS
LIN {X 0.027,Y -520.698,Z 730.155,A 0.000,B 0.000,C 90.000,E1 243.819} C_DIS
LIN {X -0.107,Y -518.624,Z 730.148,A 0.000,B 0.000,C 90.000,E1 242.666} C_DIS
LIN {X 0.087,Y -515.746,Z 730.140,A 0.000,B 0.000,C 90.000,E1 241.179} C_DIS
LIN {X -0.233,Y -512.885,Z 730.132,A 0.000,B 0.000,C 90.000,E1 239.744} C_DIS
LIN {X -0.083,Y -509.855,Z 730.124,A 0.000,B 0.000,C 90.000,E1 238.250} C_DIS
LIN {X 0.017,Y -506.763,Z 730.115,A 0.000,B 0.000,C 90.000,E1 236.755} C_DIS
LIN {X -0.150,Y -504.878,Z 730.110,A 0.000,B 0.000,C 90.000,E1 235.881} C_DIS
LIN {X -0.172,Y -502.141,Z 730.104,A 0.000,B 0.000,C 90.000,E1 234.689} C_DIS
LIN {X -0.234,Y -499.278,Z 730.097,A 0.000,B 0.000,C 90.000,E1 233.497} C_DIS
LIN {X -0.178,Y -495.451,Z 730.089,A 0.000,B 0.000,C 90.000,E1 231.984} C_DIS
LIN {X -0.041,Y -489.527,Z 730.075,A 0.000,B 0.000,C 90.000,E1 229.542} C_DIS
LIN {X -0.097,Y -485.335,Z 730.065,A 0.000,B 0.000,C 90.000,E1 227.715} C_DIS
LIN {X -0.276,Y -481.240,Z 730.055,A 0.000,B 0.000,C 90.000,E1 225.891} C_DIS
LIN {X -0.092,Y -476.532,Z 730.043,A 0.000,B 0.000,C 90.000,E1 223.704} C_DIS
LIN {X -0.118,Y -472.621,Z 730.032,A 0.000,B 0.000,C 90.000,E1 221.838} C_DIS
LIN {X 0.272,Y -469.897,Z 730.025,A 0.000,B 0.000,C 90.000,E1 220.539} C_DIS
LIN {X 0.077,Y -466.435,Z 730.017,A 0.000,B 0.000,C 90.000,E1 218.991} C_DIS
LIN {X -0.180,Y -462.927,Z 730.008,A 0.000,B 0.000,C 90.000,E1 217.443} C_DIS
LIN {X 0.082,Y -458.266,Z 729.996,A 0.000,B 0.000,C 90.000,E1 215.185} C_DIS
LIN {X 0.056,Y -453.324,Z 729.981,A 0.000,B 0.000,C 90.000,E1 212.625} C_DIS
LIN {X -0.078,Y -449.161,Z 729.969,A 0.000,B 0.000,C 90.000,E1 210.384} C_DIS
LIN {X -0.007,Y -444.934,Z 729.956,A 0.000,B 0.000,C 90.000,E1 208.103} C_DIS
LIN {X -0.142,Y -441.947,Z 729.947,A 0.000,B 0.000,C 90.000,E1 206.488} C_DIS
LIN {X -0.107,Y -438.276,Z 729.936,A 0.000,B 0.000,C 90.000,E1 204.515} C_DIS
LIN {X 0.223,Y -435.248,Z 729.927,A 0.000,B 0.000,C 90.000,E1 202.823} C_DIS
LIN {X -0.241,Y -432.142,Z 729.918,A 0.000,B 0.000,C 90.000,E1 201.227} C_DIS
LIN {X 0.054,Y -429.077,Z 729.909,A 0.000,B 0.000,C 90.000,E1 199.523} C_DIS
LIN {X -0.124,Y -426.029,Z 729.899,A 0.000,B 0.000,C 90.000,E1 197.873} C_DIS
LIN {X -0.221,Y -422.774,Z 729.890,A 0.000,B 0.000,C 90.000,E1 196.205} C_DIS
LIN {X -0.153,Y -418.458,Z 729.877,A 0.000,B 0.000,C 90.000,E1 193.828} C_DIS
LIN {X -0.050,Y -414.860,Z 729.865,A 0.000,B 0.000,C 90.000,E1 191.771} C_DIS
LIN {X -0.031,Y -409.479,Z 729.848,A 0.000,B 0.000,C 90.000,E1 188.681} C_DIS
LIN {X -0.017,Y -406.166,Z 729.837,A 0.000,B 0.000,C 90.000,E1 186.606} C_DIS
LIN {X -0.071,Y -403.541,Z 729.827,A 0.000,B 0.000,C 90.000,E1 184.878} C_DIS
LIN {X 0.044,Y -399.237,Z 729.810,A 0.000,B 0.000,C 90.000,E1 181.718} C_DIS
LIN {X 0.009,Y -396.013,Z 729.794,A 0.000,B 0.000,C 90.000,E1 178.912} C_DIS
LIN {X 0.042,Y -393.931,Z 729.782,A 0.000,B 0.000,C 90.000,E1 176.788} C_DIS
LIN {X -0.169,Y -391.246,Z 729.765,A 0.000,B 0.000,C 90.000,E1 173.628} C_DIS
LIN {X -0.026,Y -389.078,Z 729.743,A 0.000,B 0.000,C 90.000,E1 169.690} C_DIS
LIN {X -0.183,Y -388.538,Z 729.735,A 0.000,B 0.000,C 90.000,E1 168.285} C_DIS
LIN {X 0.011,Y -387.666,Z 729.721,A 0.000,B 0.000,C 90.000,E1 165.755} C_DIS
LIN {X -0.024,Y -386.948,Z 729.701,A 0.000,B 0.000,C 90.000,E1 162.181} C_DIS
LIN {X -0.194,Y -386.607,Z 729.687,A 0.000,B 0.000,C 90.000,E1 159.699} C_DIS
LIN {X -0.112,Y -386.355,Z 729.673,A 0.000,B 0.000,C 90.000,E1 157.177} C_DIS
LIN {X -0.102,Y -386.351,Z 729.661,A 0.000,B 0.000,C 90.000,E1 155.025} C_DIS
LIN {X 0.089,Y -386.616,Z 729.647,A 0.000,B 0.000,C 90.000,E1 152.487} C_DIS
LIN {X 0.115,Y -387.189,Z 729.635,A 0.000,B 0.000,C 90.000,E1 150.333} C_DIS
LIN {X -0.131,Y -389.867,Z 729.609,A 0.000,B 0.000,C 90.000,E1 145.722} C_DIS
LIN {X 0.162,Y -393.221,Z 729.592,A 0.000,B 0.000,C 90.000,E1 142.477} C_DIS
LIN {X -0.133,Y -394.708,Z 729.586,A 0.000,B 0.000,C 90.000,E1 141.457} C_DIS
LIN {X 0.050,Y -395.674,Z 729.582,A 0.000,B 0.000,C 90.000,E1 140.723} C_DIS
LIN {X 0.035,Y -397.608,Z 729.576,A 0.000,B 0.000,C 90.000,E1 139.666} C_DIS
LIN {X -0.061,Y -399.164,Z 729.572,A 0.000,B 0.000,C 90.000,E1 138.976} C_DIS
LIN {X 0.254,Y -401.191,Z 729.568,A 0.000,B 0.000,C 90.000,E1 138.243} C_DIS
LIN {X 0.187,Y -404.100,Z 729.564,A 0.000,B 0.000,C 90.000,E1 137.553} C_DIS
LIN {X 0.137,Y -406.418,Z 729.562,A 0.000,B 0.000,C 90.000,E1 137.148} C_DIS
LIN {X 0.019,Y -410.644,Z 729.559,A 0.000,B 0.000,C 90.000,E1 136.581} C_DIS
LIN {X -0.182,Y -416.386,Z 729.555,A 0.000,B 0.000,C 90.000,E1 135.972} C_DIS
LIN {X -0.142,Y -436.769,Z 729.544,A 0.000,B 0.000,C 90.000,E1 133.947} C_DIS
LIN {X 0.126,Y -445.491,Z 729.540,A 0.000,B 0.000,C 90.000,E1 133.095} C_DIS
LIN {X -0.042,Y -454.413,Z 729.535,A 0.000,B 0.000,C 90.000,E1 132.285} C_DIS
LIN {X 0.147,Y -466.020,Z 729.529,A 0.000,B 0.000,C 90.000,E1 131.148} C_DIS
LIN {X -0.114,Y -474.533,Z 729.524,A 0.000,B 0.000,C 90.000,E1 130.334} C_DIS
LIN {X -0.089,Y -480.107,Z 729.521,A 0.000,B 0.000,C 90.000,E1 129.769} C_DIS
LIN {X 0.023,Y -489.612,Z 729.515,A 0.000,B 0.000,C 90.000,E1 128.749} C_DIS
LIN {X -0.051,Y -494.907,Z 729.512,A 0.000,B 0.000,C 90.000,E1 128.177} C_DIS
LIN {X -0.049,Y -498.748,Z 729.510,A 0.000,B 0.000,C 90.000,E1 127.729} C_DIS
LIN {X -0.075,Y -502.414,Z 729.507,A 0.000,B 0.000,C 90.000,E1 127.282} C_DIS
LIN {X 0.098,Y -510.345,Z 729.501,A 0.000,B 0.000,C 90.000,E1 126.217} C_DIS
LIN {X -0.270,Y -515.450,Z 729.497,A 0.000,B 0.000,C 90.000,E1 125.518} C_DIS
LIN {X 0.130,Y -519.935,Z 729.493,A 0.000,B 0.000,C 90.000,E1 124.739} C_DIS
LIN {X -0.105,Y -522.600,Z 729.491,A 0.000,B 0.000,C 90.000,E1 124.326} C_DIS
LIN {X -0.095,Y -527.210,Z 729.486,A 0.000,B 0.000,C 90.000,E1 123.452} C_DIS
LIN {X -0.316,Y -530.776,Z 729.482,A 0.000,B 0.000,C 90.000,E1 122.752} C_DIS
LIN {X -0.063,Y -534.063,Z 729.478,A 0.000,B 0.000,C 90.000,E1 122.005} C_DIS
LIN {X 0.079,Y -537.782,Z 729.473,A 0.000,B 0.000,C 90.000,E1 121.131} C_DIS
LIN {X -0.013,Y -542.465,Z 729.467,A 0.000,B 0.000,C 90.000,E1 120.001} C_DIS
LIN {X -0.056,Y -545.868,Z 729.462,A 0.000,B 0.000,C 90.000,E1 119.155} C_DIS
LIN {X -0.042,Y -550.083,Z 729.456,A 0.000,B 0.000,C 90.000,E1 118.025} C_DIS
LIN {X -0.006,Y -553.006,Z 729.451,A 0.000,B 0.000,C 90.000,E1 117.180} C_DIS
LIN {X -0.189,Y -555.732,Z 729.446,A 0.000,B 0.000,C 90.000,E1 116.360} C_DIS
LIN {X -0.098,Y -558.114,Z 729.442,A 0.000,B 0.000,C 90.000,E1 115.515} C_DIS
LIN {X 0.283,Y -560.167,Z 729.437,A 0.000,B 0.000,C 90.000,E1 114.643} C_DIS
LIN {X 0.181,Y -561.984,Z 729.432,A 0.000,B 0.000,C 90.000,E1 113.823} C_DIS
LIN {X -0.127,Y -563.562,Z 729.428,A 0.000,B 0.000,C 90.000,E1 113.025} C_DIS
LIN {X -0.198,Y -564.885,Z 729.423,A 0.000,B 0.000,C 90.000,E1 112.206} C_DIS
LIN {X 0.195,Y -567.027,Z 729.416,A 0.000,B 0.000,C 90.000,E1 110.791} C_DIS
LIN {X -0.105,Y -569.102,Z 729.408,A 0.000,B 0.000,C 90.000,E1 109.450} C_DIS
LIN {X -0.208,Y -571.384,Z 729.399,A 0.000,B 0.000,C 90.000,E1 107.819} C_DIS
LIN {X 0.117,Y -573.502,Z 729.390,A 0.000,B 0.000,C 90.000,E1 106.150} C_DIS
LIN {X 0.139,Y -575.905,Z 729.379,A 0.000,B 0.000,C 90.000,E1 104.245} C_DIS
LIN {X -0.152,Y -577.862,Z 729.370,A 0.000,B 0.000,C 90.000,E1 102.647} C_DIS
LIN {X 0.150,Y -579.223,Z 729.364,A 0.000,B 0.000,C 90.000,E1 101.535} C_DIS
LIN {X 0.249,Y -581.230,Z 729.355,A 0.000,B 0.000,C 90.000,E1 99.905} C_DIS
LIN {X -0.076,Y -582.444,Z 729.349,A 0.000,B 0.000,C 90.000,E1 98.859} C_DIS
LIN {X -0.235,Y -583.844,Z 729.342,A 0.000,B 0.000,C 90.000,E1 97.530} C_DIS
LIN {X 0.036,Y -585.714,Z 729.331,A 0.000,B 0.000,C 90.000,E1 95.625} C_DIS
LIN {X -0.130,Y -587.014,Z 729.324,A 0.000,B 0.000,C 90.000,E1 94.302} C_DIS
LIN {X -0.088,Y -588.381,Z 729.315,A 0.000,B 0.000,C 90.000,E1 92.694} C_DIS
LIN {X 0.136,Y -589.158,Z 729.309,A 0.000,B 0.000,C 90.000,E1 91.604} C_DIS
LIN {X 0.175,Y -590.122,Z 729.300,A 0.000,B 0.000,C 90.000,E1 90.000} C_DIS
LIN {X 0.027,Y -590.774,Z 729.293,A 0.000,B 0.000,C 90.000,E1 88.682} C_DIS
LIN {X -0.098,Y -591.244,Z 729.285,A 0.000,B 0.000,C 90.000,E1 87.364} C_DIS
LIN {X -0.217,Y -591.561,Z 729.278,A 0.000,B 0.000,C 90.000,E1 86.045} C_DIS
LIN {X -0.293,Y -591.797,Z 729.271,A 0.000,B 0.000,C 90.000,E1 84.723} C_DIS
LIN {X -0.170,Y -591.860,Z 729.266,A 0.000,B 0.000,C 90.000,E1 83.913} C_DIS
LIN {X 0.022,Y -591.887,Z 729.257,A 0.000,B 0.000,C 90.000,E1 82.299} C_DIS
LIN {X -0.163,Y -591.758,Z 729.251,A 0.000,B 0.000,C 90.000,E1 81.254} C_DIS
LIN {X -0.177,Y -591.459,Z 729.244,A 0.000,B 0.000,C 90.000,E1 79.926} C_DIS
LIN {X 0.006,Y -590.834,Z 729.237,A 0.000,B 0.000,C 90.000,E1 78.578} C_DIS
LIN {X -0.122,Y -589.985,Z 729.228,A 0.000,B 0.000,C 90.000,E1 76.992} C_DIS
LIN {X 0.130,Y -588.811,Z 729.217,A 0.000,B 0.000,C 90.000,E1 75.102} C_DIS
LIN {X -0.155,Y -587.779,Z 729.210,A 0.000,B 0.000,C 90.000,E1 73.795} C_DIS
LIN {X -0.143,Y -586.926,Z 729.204,A 0.000,B 0.000,C 90.000,E1 72.725} C_DIS
LIN {X 0.030,Y -585.970,Z 729.198,A 0.000,B 0.000,C 90.000,E1 71.638} C_DIS
LIN {X 0.049,Y -584.650,Z 729.191,A 0.000,B 0.000,C 90.000,E1 70.296} C_DIS
LIN {X -0.223,Y -583.781,Z 729.186,A 0.000,B 0.000,C 90.000,E1 69.518} C_DIS
LIN {X -0.037,Y -582.175,Z 729.179,A 0.000,B 0.000,C 90.000,E1 68.156} C_DIS
LIN {X 0.263,Y -580.785,Z 729.173,A 0.000,B 0.000,C 90.000,E1 67.050} C_DIS
LIN {X -0.142,Y -578.738,Z 729.165,A 0.000,B 0.000,C 90.000,E1 65.741} C_DIS
LIN {X -0.196,Y -576.873,Z 729.159,A 0.000,B 0.000,C 90.000,E1 64.665} C_DIS
LIN {X -0.125,Y -575.304,Z 729.155,A 0.000,B 0.000,C 90.000,E1 63.845} C_DIS
LIN {X 0.028,Y -572.963,Z 729.149,A 0.000,B 0.000,C 90.000,E1 62.743} C_DIS
LIN {X 0.316,Y -570.983,Z 729.144,A 0.000,B 0.000,C 90.000,E1 61.897} C_DIS
LIN {X -0.088,Y -568.098,Z 729.138,A 0.000,B 0.000,C 90.000,E1 60.845} C_DIS
LIN {X -0.041,Y -564.847,Z 729.132,A 0.000,B 0.000,C 90.000,E1 59.744} C_DIS
LIN {X -0.044,Y -562.128,Z 729.127,A 0.000,B 0.000,C 90.000,E1 58.918} C_DIS
LIN {X 0.114,Y -559.250,Z 729.123,A 0.000,B 0.000,C 90.000,E1 58.074} C_DIS
LIN {X -0.020,Y -557.176,Z 729.120,A 0.000,B 0.000,C 90.000,E1 57.533} C_DIS
LIN {X -0.096,Y -553.677,Z 729.115,A 0.000,B 0.000,C 90.000,E1 56.707} C_DIS
LIN {X -0.088,Y -550.405,Z 729.111,A 0.000,B 0.000,C 90.000,E1 56.008} C_DIS
LIN {X -0.055,Y -546.943,Z 729.107,A 0.000,B 0.000,C 90.000,E1 55.308} C_DIS
LIN {X -0.245,Y -542.144,Z 729.103,A 0.000,B 0.000,C 90.000,E1 54.482} C_DIS
LIN {X -0.044,Y -539.661,Z 729.100,A 0.000,B 0.000,C 90.000,E1 54.036} C_DIS
LIN {X -0.005,Y -536.082,Z 729.097,A 0.000,B 0.000,C 90.000,E1 53.463} C_DIS
LIN {X -0.152,Y -530.954,Z 729.093,A 0.000,B 0.000,C 90.000,E1 52.763} C_DIS
LIN {X -0.008,Y -527.708,Z 729.091,A 0.000,B 0.000,C 90.000,E1 52.316} C_DIS
LIN {X -0.051,Y -522.654,Z 729.087,A 0.000,B 0.000,C 90.000,E1 51.743} C_DIS
LIN {X -0.189,Y -518.671,Z 729.085,A 0.000,B 0.000,C 90.000,E1 51.331} C_DIS
LIN {X -0.323,Y -512.808,Z 729.082,A 0.000,B 0.000,C 90.000,E1 50.803} C_DIS
LIN {X -0.126,Y -506.825,Z 729.079,A 0.000,B 0.000,C 90.000,E1 50.275} C_DIS
LIN {X -0.109,Y -502.181,Z 729.077,A 0.000,B 0.000,C 90.000,E1 49.908} C_DIS
LIN {X -0.171,Y -495.777,Z 729.075,A 0.000,B 0.000,C 90.000,E1 49.461} C_DIS
LIN {X -0.188,Y -487.540,Z 729.072,A 0.000,B 0.000,C 90.000,E1 48.933} C_DIS
LIN {X -0.060,Y -478.094,Z 729.068,A 0.000,B 0.000,C 90.000,E1 48.324} C_DIS
LIN {X -0.023,Y -464.925,Z 729.064,A 0.000,B 0.000,C 90.000,E1 47.514} C_DIS
LIN {X -0.110,Y -450.678,Z 729.059,A 0.000,B 0.000,C 90.000,E1 46.620} C_DIS
LIN {X 0.194,Y -423.575,Z 729.049,A 0.000,B 0.000,C 90.000,E1 44.757} C_DIS
LIN {X 0.108,Y -417.356,Z 729.046,A 0.000,B 0.000,C 90.000,E1 44.271} C_DIS
LIN {X 0.078,Y -417.332,Z 729.046,A 0.000,B 0.000,C 90.000,E1 44.271} C_DIS
LIN {X 0.169,Y -408.314,Z 729.022,A 0.000,B 0.000,C 90.000,E1 39.930} C_DIS
LIN {X 0.193,Y -406.005,Z 729.014,A 0.000,B 0.000,C 90.000,E1 38.543} C_DIS
LIN {X -0.002,Y -404.890,Z 729.011,A 0.000,B 0.000,C 90.000,E1 38.051} C_DIS
LIN {X -0.026,Y -405.444,Z 728.991,A 0.000,B 0.000,C 90.000,E1 34.405} C_DIS
LIN {X 0.105,Y -406.422,Z 728.978,A 0.000,B 0.000,C 90.000,E1 31.957} C_DIS
LIN {X 0.136,Y -407.352,Z 728.966,A 0.000,B 0.000,C 90.000,E1 29.873} C_DIS
LIN {X -0.220,Y -408.544,Z 728.955,A 0.000,B 0.000,C 90.000,E1 27.847} C_DIS
LIN {X -0.092,Y -410.023,Z 728.941,A 0.000,B 0.000,C 90.000,E1 25.412} C_DIS
LIN {X 0.015,Y -412.217,Z 728.926,A 0.000,B 0.000,C 90.000,E1 22.642} C_DIS
LIN {X 0.067,Y -413.814,Z 728.916,A 0.000,B 0.000,C 90.000,E1 20.918} C_DIS
LIN {X -0.084,Y -416.309,Z 728.903,A 0.000,B 0.000,C 90.000,E1 18.544} C_DIS
LIN {X -0.067,Y -418.850,Z 728.892,A 0.000,B 0.000,C 90.000,E1 16.496} C_DIS
LIN {X 0.011,Y -422.562,Z 728.877,A 0.000,B 0.000,C 90.000,E1 13.772} C_DIS
LIN {X -0.159,Y -425.471,Z 728.865,A 0.000,B 0.000,C 90.000,E1 11.771} C_DIS
LIN {X -0.037,Y -428.001,Z 728.856,A 0.000,B 0.000,C 90.000,E1 10.074} C_DIS
LIN {X 0.212,Y -431.519,Z 728.843,A 0.000,B 0.000,C 90.000,E1 7.701} C_DIS
LIN {X 0.075,Y -435.021,Z 728.830,A 0.000,B 0.000,C 90.000,E1 5.391} C_DIS
LIN {X -0.055,Y -438.848,Z 728.817,A 0.000,B 0.000,C 90.000,E1 3.094} C_DIS
LIN {X 0.004,Y -443.502,Z 728.803,A 0.000,B 0.000,C 90.000,E1 0.458} C_DIS
LIN {X -0.017,Y -447.955,Z 728.790,A 0.000,B 0.000,C 90.000,E1 358.165} C_DIS
LIN {X 0.072,Y -453.915,Z 728.774,A 0.000,B 0.000,C 90.000,E1 355.241} C_DIS
LIN {X 0.123,Y -457.415,Z 728.765,A 0.000,B 0.000,C 90.000,E1 353.628} C_DIS
LIN {X -0.154,Y -460.816,Z 728.756,A 0.000,B 0.000,C 90.000,E1 352.064} C_DIS
LIN {X -0.108,Y -464.739,Z 728.745,A 0.000,B 0.000,C 90.000,E1 350.151} C_DIS
LIN {X 0.024,Y -467.266,Z 728.738,A 0.000,B 0.000,C 90.000,E1 348.870} C_DIS
LIN {X 0.006,Y -470.201,Z 728.729,A 0.000,B 0.000,C 90.000,E1 347.297} C_DIS
LIN {X 0.075,Y -473.638,Z 728.719,A 0.000,B 0.000,C 90.000,E1 345.408} C_DIS
LIN {X -0.140,Y -477.712,Z 728.707,A 0.000,B 0.000,C 90.000,E1 343.251} C_DIS
LIN {X -0.068,Y -480.981,Z 728.698,A 0.000,B 0.000,C 90.000,E1 341.692} C_DIS
LIN {X -0.238,Y -482.597,Z 728.695,A 0.000,B 0.000,C 90.000,E1 341.094} C_DIS
LIN {X 0.216,Y -484.592,Z 728.691,A 0.000,B 0.000,C 90.000,E1 340.423} C_DIS
LIN {X -0.151,Y -486.641,Z 728.689,A 0.000,B 0.000,C 90.000,E1 340.007} C_DIS
LIN {X -0.137,Y -488.336,Z 728.687,A 0.000,B 0.000,C 90.000,E1 339.699} C_DIS
LIN {X -0.195,Y -490.886,Z 728.685,A 0.000,B 0.000,C 90.000,E1 339.337} C_DIS
LIN {X 0.141,Y -494.895,Z 728.683,A 0.000,B 0.000,C 90.000,E1 338.847} C_DIS
LIN {X -0.010,Y -496.431,Z 728.682,A 0.000,B 0.000,C 90.000,E1 338.720} C_DIS
LIN {X 0.263,Y -503.113,Z 728.679,A 0.000,B 0.000,C 90.000,E1 338.156} C_DIS
LIN {X -0.053,Y -523.608,Z 728.672,A 0.000,B 0.000,C 90.000,E1 336.869} C_DIS
LIN {X -0.110,Y -533.232,Z 728.668,A 0.000,B 0.000,C 90.000,E1 336.282} C_DIS
LIN {X -0.011,Y -539.441,Z 728.666,A 0.000,B 0.000,C 90.000,E1 335.869} C_DIS
LIN {X 0.171,Y -546.744,Z 728.663,A 0.000,B 0.000,C 90.000,E1 335.305} C_DIS
LIN {X 0.077,Y -550.974,Z 728.661,A 0.000,B 0.000,C 90.000,E1 334.973} C_DIS
LIN {X -0.187,Y -558.934,Z 728.657,A 0.000,B 0.000,C 90.000,E1 334.280} C_DIS
LIN {X -0.172,Y -565.510,Z 728.654,A 0.000,B 0.000,C 90.000,E1 333.640} C_DIS
LIN {X 0.075,Y -573.093,Z 728.649,A 0.000,B 0.000,C 90.000,E1 332.820} C_DIS
LIN {X -0.035,Y -579.119,Z 728.645,A 0.000,B 0.000,C 90.000,E1 332.153} C_DIS
LIN {X -0.244,Y -584.884,Z 728.642,A 0.000,B 0.000,C 90.000,E1 331.513} C_DIS
LIN {X 0.245,Y -590.435,Z 728.638,A 0.000,B 0.000,C 90.000,E1 330.795} C_DIS
LIN {X 0.181,Y -597.809,Z 728.633,A 0.000,B 0.000,C 90.000,E1 329.871} C_DIS
LIN {X 0.237,Y -603.878,Z 728.628,A 0.000,B 0.000,C 90.000,E1 329.076} C_DIS
LIN {X -0.193,Y -610.617,Z 728.623,A 0.000,B 0.000,C 90.000,E1 328.201} C_DIS
LIN {X 0.320,Y -616.038,Z 728.619,A 0.000,B 0.000,C 90.000,E1 327.375} C_DIS
LIN {X 0.027,Y -622.017,Z 728.614,A 0.000,B 0.000,C 90.000,E1 326.501} C_DIS
LIN {X -0.196,Y -626.012,Z 728.610,A 0.000,B 0.000,C 90.000,E1 325.881} C_DIS
LIN {X -0.034,Y -632.123,Z 728.605,A 0.000,B 0.000,C 90.000,E1 324.848} C_DIS
LIN {X 0.193,Y -636.482,Z 728.601,A 0.000,B 0.000,C 90.000,E1 324.069} C_DIS
LIN {X -0.148,Y -642.524,Z 728.594,A 0.000,B 0.000,C 90.000,E1 322.970} C_DIS
LIN {X 0.190,Y -646.374,Z 728.590,A 0.000,B 0.000,C 90.000,E1 322.190} C_DIS
LIN {X -0.005,Y -651.798,Z 728.584,A 0.000,B 0.000,C 90.000,E1 321.090} C_DIS
LIN {X 0.313,Y -657.407,Z 728.577,A 0.000,B 0.000,C 90.000,E1 319.828} C_DIS
LIN {X 0.245,Y -661.537,Z 728.572,A 0.000,B 0.000,C 90.000,E1 318.852} C_DIS
LIN {X -0.271,Y -665.478,Z 728.566,A 0.000,B 0.000,C 90.000,E1 317.919} C_DIS
LIN {X 0.209,Y -669.008,Z 728.561,A 0.000,B 0.000,C 90.000,E1 316.905} C_DIS
LIN {X -0.215,Y -672.349,Z 728.555,A 0.000,B 0.000,C 90.000,E1 315.972} C_DIS
LIN {X -0.157,Y -674.737,Z 728.551,A 0.000,B 0.000,C 90.000,E1 315.243} C_DIS
LIN {X -0.041,Y -677.748,Z 728.546,A 0.000,B 0.000,C 90.000,E1 314.271} C_DIS
LIN {X 0.151,Y -681.235,Z 728.539,A 0.000,B 0.000,C 90.000,E1 313.056} C_DIS
LIN {X 0.432,Y -684.440,Z 728.533,A 0.000,B 0.000,C 90.000,E1 311.838} C_DIS
LIN {X 0.197,Y -686.750,Z 728.527,A 0.000,B 0.000,C 90.000,E1 310.906} C_DIS
LIN {X 0.064,Y -688.950,Z 728.522,A 0.000,B 0.000,C 90.000,E1 309.967} C_DIS
LIN {X -0.128,Y -690.753,Z 728.517,A 0.000,B 0.000,C 90.000,E1 309.036} C_DIS
LIN {X -0.202,Y -692.348,Z 728.512,A 0.000,B 0.000,C 90.000,E1 308.096} C_DIS
LIN {X 0.361,Y -694.016,Z 728.505,A 0.000,B 0.000,C 90.000,E1 306.870} C_DIS
LIN {X -0.024,Y -695.462,Z 728.499,A 0.000,B 0.000,C 90.000,E1 305.724} C_DIS
LIN {X 0.123,Y -696.427,Z 728.493,A 0.000,B 0.000,C 90.000,E1 304.771} C_DIS
LIN {X -0.001,Y -697.590,Z 728.485,A 0.000,B 0.000,C 90.000,E1 303.372} C_DIS
LIN {X -0.155,Y -698.602,Z 728.479,A 0.000,B 0.000,C 90.000,E1 302.212} C_DIS
LIN {X -0.042,Y -699.722,Z 728.471,A 0.000,B 0.000,C 90.000,E1 300.797} C_DIS
LIN {X 0.146,Y -700.087,Z 728.467,A 0.000,B 0.000,C 90.000,E1 300.079} C_DIS
LIN {X -0.069,Y -700.455,Z 728.459,A 0.000,B 0.000,C 90.000,E1 298.693} C_DIS
LIN {X 0.056,Y -700.788,Z 728.453,A 0.000,B 0.000,C 90.000,E1 297.513} C_DIS
LIN {X 0.027,Y -701.679,Z 728.441,A 0.000,B 0.000,C 90.000,E1 295.412} C_DIS
LIN {X 0.304,Y -701.770,Z 728.440,A 0.000,B 0.000,C 90.000,E1 295.155} C_DIS
LIN {X -0.074,Y -701.665,Z 728.437,A 0.000,B 0.000,C 90.000,E1 294.719} C_DIS
LIN {X 0.202,Y -701.422,Z 728.436,A 0.000,B 0.000,C 90.000,E1 294.463} C_DIS
LIN {X -0.175,Y -699.995,Z 728.433,A 0.000,B 0.000,C 90.000,E1 294.027} C_DIS
LIN {X 0.097,Y -698.940,Z 728.432,A 0.000,B 0.000,C 90.000,E1 293.770} C_DIS
LIN {X 0.230,Y -697.963,Z 728.432,A 0.000,B 0.000,C 90.000,E1 293.643} C_DIS
LIN {X -0.139,Y -695.533,Z 728.430,A 0.000,B 0.000,C 90.000,E1 293.439} C_DIS
LIN {X -0.031,Y -692.814,Z 728.429,A 0.000,B 0.000,C 90.000,E1 293.206} C_DIS
LIN {X 0.214,Y -691.107,Z 728.428,A 0.000,B 0.000,C 90.000,E1 293.078} C_DIS
LIN {X 0.160,Y -686.388,Z 728.427,A 0.000,B 0.000,C 90.000,E1 292.898} C_DIS
LIN {X 0.170,Y -682.038,Z 728.427,A 0.000,B 0.000,C 90.000,E1 292.770} C_DIS
LIN {X 0.095,Y -676.661,Z 728.426,A 0.000,B 0.000,C 90.000,E1 292.642} C_DIS
LIN {X -0.197,Y -655.029,Z 728.424,A 0.000,B 0.000,C 90.000,E1 292.386} C_DIS
LIN {X 0.021,Y -645.184,Z 728.423,A 0.000,B 0.000,C 90.000,E1 292.206} C_DIS
LIN {X -0.111,Y -631.816,Z 728.422,A 0.000,B 0.000,C 90.000,E1 291.950} C_DIS
LIN {X 0.301,Y -618.434,Z 728.420,A 0.000,B 0.000,C 90.000,E1 291.589} C_DIS
LIN {X -0.169,Y -594.398,Z 728.416,A 0.000,B 0.000,C 90.000,E1 290.972} C_DIS
LIN {X 0.146,Y -576.795,Z 728.414,A 0.000,B 0.000,C 90.000,E1 290.429} C_DIS
LIN {X 0.212,Y -567.694,Z 728.412,A 0.000,B 0.000,C 90.000,E1 290.174} C_DIS
LIN {X -0.229,Y -561.117,Z 728.411,A 0.000,B 0.000,C 90.000,E1 289.993} C_DIS
LIN {X -0.031,Y -556.594,Z 728.409,A 0.000,B 0.000,C 90.000,E1 289.704} C_DIS
LIN {X -0.059,Y -556.569,Z 728.409,A 0.000,B 0.000,C 90.000,E1 289.704} C_DIS
LIN {X 0.078,Y -555.532,Z 728.408,A 0.000,B 0.000,C 90.000,E1 289.504} C_DIS
LIN {X 0.065,Y -554.876,Z 728.406,A 0.000,B 0.000,C 90.000,E1 289.087} C_DIS
LIN {X -0.155,Y -554.476,Z 728.400,A 0.000,B 0.000,C 90.000,E1 288.000} C_DIS
LIN {X 0.063,Y -553.740,Z 728.389,A 0.000,B 0.000,C 90.000,E1 286.024} C_DIS
LIN {X 0.229,Y -552.946,Z 728.377,A 0.000,B 0.000,C 90.000,E1 283.772} C_DIS
LIN {X -0.004,Y -552.416,Z 728.367,A 0.000,B 0.000,C 90.000,E1 282.119} C_DIS
LIN {X 0.063,Y -551.749,Z 728.358,A 0.000,B 0.000,C 90.000,E1 280.433} C_DIS
LIN {X 0.098,Y -551.116,Z 728.350,A 0.000,B 0.000,C 90.000,E1 279.029} C_DIS
LIN {X 0.087,Y -550.177,Z 728.339,A 0.000,B 0.000,C 90.000,E1 277.068} C_DIS
LIN {X 0.018,Y -549.503,Z 728.330,A 0.000,B 0.000,C 90.000,E1 275.391} C_DIS
LIN {X 0.242,Y -549.130,Z 728.324,A 0.000,B 0.000,C 90.000,E1 274.245} C_DIS
LIN {X 0.046,Y -548.394,Z 728.314,A 0.000,B 0.000,C 90.000,E1 272.579} C_DIS
LIN {X -0.244,Y -547.820,Z 728.307,A 0.000,B 0.000,C 90.000,E1 271.203} C_DIS
LIN {X -0.008,Y -546.982,Z 728.299,A 0.000,B 0.000,C 90.000,E1 269.771} C_DIS
LIN {X 0.210,Y -546.114,Z 728.291,A 0.000,B 0.000,C 90.000,E1 268.339} C_DIS
LIN {X -0.059,Y -545.070,Z 728.282,A 0.000,B 0.000,C 90.000,E1 266.674} C_DIS
LIN {X 0.202,Y -543.881,Z 728.272,A 0.000,B 0.000,C 90.000,E1 264.951} C_DIS
LIN {X -0.134,Y -542.869,Z 728.264,A 0.000,B 0.000,C 90.000,E1 263.571} C_DIS
LIN {X 0.102,Y -541.981,Z 728.258,A 0.000,B 0.000,C 90.000,E1 262.413} C_DIS
LIN {X -0.063,Y -540.315,Z 728.247,A 0.000,B 0.000,C 90.000,E1 260.443} C_DIS
LIN {X -0.256,Y -538.814,Z 728.237,A 0.000,B 0.000,C 90.000,E1 258.757} C_DIS
LIN {X 0.077,Y -537.685,Z 728.230,A 0.000,B 0.000,C 90.000,E1 257.297} C_DIS
LIN {X -0.018,Y -536.403,Z 728.222,A 0.000,B 0.000,C 90.000,E1 255.880} C_DIS
LIN {X -0.185,Y -535.232,Z 728.215,A 0.000,B 0.000,C 90.000,E1 254.755} C_DIS
LIN {X -0.181,Y -533.721,Z 728.207,A 0.000,B 0.000,C 90.000,E1 253.323} C_DIS
LIN {X -0.018,Y -531.940,Z 728.198,A 0.000,B 0.000,C 90.000,E1 251.583} C_DIS
LIN {X -0.120,Y -530.946,Z 728.193,A 0.000,B 0.000,C 90.000,E1 250.732} C_DIS
LIN {X 0.142,Y -528.989,Z 728.185,A 0.000,B 0.000,C 90.000,E1 249.263} C_DIS
LIN {X 0.188,Y -527.443,Z 728.179,A 0.000,B 0.000,C 90.000,E1 248.103} C_DIS
LIN {X 0.261,Y -524.888,Z 728.169,A 0.000,B 0.000,C 90.000,E1 246.357} C_DIS
LIN {X -0.042,Y -523.033,Z 728.162,A 0.000,B 0.000,C 90.000,E1 245.229} C_DIS
LIN {X 0.000,Y -520.658,Z 728.154,A 0.000,B 0.000,C 90.000,E1 243.768} C_DIS
LIN {X -0.139,Y -518.553,Z 728.148,A 0.000,B 0.000,C 90.000,E1 242.615} C_DIS
LIN {X 0.047,Y -515.696,Z 728.140,A 0.000,B 0.000,C 90.000,E1 241.129} C_DIS
LIN {X -0.021,Y -512.799,Z 728.132,A 0.000,B 0.000,C 90.000,E1 239.665} C_DIS
LIN {X 0.224,Y -510.379,Z 728.125,A 0.000,B 0.000,C 90.000,E1 238.456} C_DIS
LIN {X 0.004,Y -507.922,Z 728.118,A 0.000,B 0.000,C 90.000,E1 237.296} C_DIS
LIN {X 0.170,Y -505.413,Z 728.112,A 0.000,B 0.000,C 90.000,E1 236.087} C_DIS
LIN {X 0.155,Y -502.774,Z 728.105,A 0.000,B 0.000,C 90.000,E1 234.895} C_DIS
LIN {X 0.102,Y -499.887,Z 728.098,A 0.000,B 0.000,C 90.000,E1 233.703} C_DIS
LIN {X 0.302,Y -496.907,Z 728.092,A 0.000,B 0.000,C 90.000,E1 232.477} C_DIS
LIN {X 0.013,Y -490.152,Z 728.077,A 0.000,B 0.000,C 90.000,E1 229.784} C_DIS
LIN {X -0.036,Y -485.948,Z 728.066,A 0.000,B 0.000,C 90.000,E1 227.957} C_DIS
LIN {X -0.203,Y -481.783,Z 728.056,A 0.000,B 0.000,C 90.000,E1 226.134} C_DIS
LIN {X -0.123,Y -477.709,Z 728.046,A 0.000,B 0.000,C 90.000,E1 224.271} C_DIS
LIN {X -0.002,Y -475.101,Z 728.039,A 0.000,B 0.000,C 90.000,E1 223.014} C_DIS
LIN {X -0.146,Y -471.805,Z 728.030,A 0.000,B 0.000,C 90.000,E1 221.472} C_DIS
LIN {X 0.233,Y -469.101,Z 728.023,A 0.000,B 0.000,C 90.000,E1 220.172} C_DIS
LIN {X -0.101,Y -466.306,Z 728.016,A 0.000,B 0.000,C 90.000,E1 218.955} C_DIS
LIN {X -0.001,Y -462.795,Z 728.008,A 0.000,B 0.000,C 90.000,E1 217.363} C_DIS
LIN {X -0.123,Y -458.143,Z 727.995,A 0.000,B 0.000,C 90.000,E1 215.152} C_DIS
LIN {X 0.215,Y -453.212,Z 727.981,A 0.000,B 0.000,C 90.000,E1 212.546} C_DIS
LIN {X -0.240,Y -449.667,Z 727.970,A 0.000,B 0.000,C 90.000,E1 210.669} C_DIS
LIN {X -0.068,Y -446.609,Z 727.961,A 0.000,B 0.000,C 90.000,E1 209.027} C_DIS
LIN {X 0.039,Y -443.600,Z 727.952,A 0.000,B 0.000,C 90.000,E1 207.385} C_DIS
LIN {X -0.166,Y -441.211,Z 727.945,A 0.000,B 0.000,C 90.000,E1 206.104} C_DIS
LIN {X -0.150,Y -437.567,Z 727.934,A 0.000,B 0.000,C 90.000,E1 204.131} C_DIS
LIN {X 0.163,Y -435.162,Z 727.927,A 0.000,B 0.000,C 90.000,E1 202.770} C_DIS
LIN {X 0.039,Y -432.684,Z 727.919,A 0.000,B 0.000,C 90.000,E1 201.461} C_DIS
LIN {X -0.070,Y -429.610,Z 727.910,A 0.000,B 0.000,C 90.000,E1 199.812} C_DIS
LIN {X -0.174,Y -425.960,Z 727.899,A 0.000,B 0.000,C 90.000,E1 197.819} C_DIS
LIN {X -0.150,Y -422.697,Z 727.890,A 0.000,B 0.000,C 90.000,E1 196.134} C_DIS
LIN {X -0.197,Y -418.425,Z 727.876,A 0.000,B 0.000,C 90.000,E1 193.772} C_DIS
LIN {X -0.091,Y -414.815,Z 727.865,A 0.000,B 0.000,C 90.000,E1 191.715} C_DIS
LIN {X -0.070,Y -409.441,Z 727.848,A 0.000,B 0.000,C 90.000,E1 188.624} C_DIS
LIN {X -0.020,Y -406.688,Z 727.838,A 0.000,B 0.000,C 90.000,E1 186.891} C_DIS
LIN {X -0.107,Y -403.517,Z 727.827,A 0.000,B 0.000,C 90.000,E1 184.821} C_DIS
LIN {X 0.044,Y -399.707,Z 727.811,A 0.000,B 0.000,C 90.000,E1 182.007} C_DIS
LIN {X -0.024,Y -396.039,Z 727.794,A 0.000,B 0.000,C 90.000,E1 178.854} C_DIS
LIN {X 0.009,Y -393.957,Z 727.782,A 0.000,B 0.000,C 90.000,E1 176.731} C_DIS
LIN {X -0.108,Y -391.628,Z 727.766,A 0.000,B 0.000,C 90.000,E1 173.913} C_DIS
LIN {X 0.164,Y -389.804,Z 727.750,A 0.000,B 0.000,C 90.000,E1 171.027} C_DIS
LIN {X -0.154,Y -388.839,Z 727.736,A 0.000,B 0.000,C 90.000,E1 168.578} C_DIS
LIN {X -0.042,Y -387.935,Z 727.723,A 0.000,B 0.000,C 90.000,E1 166.061} C_DIS
LIN {X -0.080,Y -387.167,Z 727.703,A 0.000,B 0.000,C 90.000,E1 162.489} C_DIS
LIN {X -0.089,Y -386.820,Z 727.687,A 0.000,B 0.000,C 90.000,E1 159.625} C_DIS
LIN {X 0.010,Y -386.592,Z 727.673,A 0.000,B 0.000,C 90.000,E1 157.102} C_DIS
LIN {X -0.130,Y -386.651,Z 727.661,A 0.000,B 0.000,C 90.000,E1 154.973} C_DIS
LIN {X 0.064,Y -386.857,Z 727.649,A 0.000,B 0.000,C 90.000,E1 152.794} C_DIS
LIN {X 0.088,Y -387.443,Z 727.635,A 0.000,B 0.000,C 90.000,E1 150.284} C_DIS
LIN {X 0.205,Y -391.398,Z 727.601,A 0.000,B 0.000,C 90.000,E1 144.196} C_DIS
LIN {X -0.103,Y -393.873,Z 727.589,A 0.000,B 0.000,C 90.000,E1 142.110} C_DIS
LIN {X 0.008,Y -395.796,Z 727.582,A 0.000,B 0.000,C 90.000,E1 140.678} C_DIS
LIN {X 0.090,Y -398.324,Z 727.574,A 0.000,B 0.000,C 90.000,E1 139.256} C_DIS
LIN {X -0.110,Y -399.111,Z 727.572,A 0.000,B 0.000,C 90.000,E1 138.933} C_DIS
LIN {X -0.094,Y -400.991,Z 727.568,A 0.000,B 0.000,C 90.000,E1 138.243} C_DIS
LIN {X 0.016,Y -402.408,Z 727.566,A 0.000,B 0.000,C 90.000,E1 137.877} C_DIS
LIN {X -0.165,Y -403.646,Z 727.564,A 0.000,B 0.000,C 90.000,E1 137.553} C_DIS
LIN {X 0.193,Y -405.621,Z 727.562,A 0.000,B 0.000,C 90.000,E1 137.148} C_DIS
LIN {X 0.107,Y -406.463,Z 727.561,A 0.000,B 0.000,C 90.000,E1 136.986} C_DIS
LIN {X 0.162,Y -410.204,Z 727.558,A 0.000,B 0.000,C 90.000,E1 136.458} C_DIS
LIN {X -0.243,Y -415.813,Z 727.555,A 0.000,B 0.000,C 90.000,E1 135.891} C_DIS
LIN {X 0.146,Y -436.510,Z 727.543,A 0.000,B 0.000,C 90.000,E1 133.785} C_DIS
LIN {X -0.153,Y -445.247,Z 727.539,A 0.000,B 0.000,C 90.000,E1 133.014} C_DIS
LIN {X -0.049,Y -455.566,Z 727.534,A 0.000,B 0.000,C 90.000,E1 132.043} C_DIS
LIN {X -0.177,Y -464.333,Z 727.529,A 0.000,B 0.000,C 90.000,E1 131.229} C_DIS
LIN {X -0.119,Y -472.913,Z 727.524,A 0.000,B 0.000,C 90.000,E1 130.378} C_DIS
LIN {X -0.246,Y -479.598,Z 727.521,A 0.000,B 0.000,C 90.000,E1 129.725} C_DIS
LIN {X 0.075,Y -487.817,Z 727.516,A 0.000,B 0.000,C 90.000,E1 128.830} C_DIS
LIN {X -0.009,Y -493.196,Z 727.513,A 0.000,B 0.000,C 90.000,E1 128.257} C_DIS
LIN {X 0.026,Y -497.133,Z 727.510,A 0.000,B 0.000,C 90.000,E1 127.810} C_DIS
LIN {X -0.163,Y -502.014,Z 727.507,A 0.000,B 0.000,C 90.000,E1 127.237} C_DIS
LIN {X 0.146,Y -507.513,Z 727.503,A 0.000,B 0.000,C 90.000,E1 126.503} C_DIS
LIN {X -0.087,Y -510.838,Z 727.500,A 0.000,B 0.000,C 90.000,E1 126.091} C_DIS
LIN {X -0.111,Y -514.895,Z 727.497,A 0.000,B 0.000,C 90.000,E1 125.518} C_DIS
LIN {X -0.012,Y -519.433,Z 727.493,A 0.000,B 0.000,C 90.000,E1 124.771} C_DIS
LIN {X 0.032,Y -522.908,Z 727.490,A 0.000,B 0.000,C 90.000,E1 124.199} C_DIS
LIN {X -0.227,Y -526.827,Z 727.486,A 0.000,B 0.000,C 90.000,E1 123.499} C_DIS
LIN {X -0.011,Y -530.447,Z 727.482,A 0.000,B 0.000,C 90.000,E1 122.752} C_DIS
LIN {X 0.241,Y -533.782,Z 727.478,A 0.000,B 0.000,C 90.000,E1 122.005} C_DIS
LIN {X -0.068,Y -536.371,Z 727.475,A 0.000,B 0.000,C 90.000,E1 121.465} C_DIS
LIN {X -0.180,Y -541.093,Z 727.468,A 0.000,B 0.000,C 90.000,E1 120.335} C_DIS
LIN {X -0.230,Y -545.701,Z 727.462,A 0.000,B 0.000,C 90.000,E1 119.205} C_DIS
LIN {X 0.261,Y -549.945,Z 727.456,A 0.000,B 0.000,C 90.000,E1 118.025} C_DIS
LIN {X -0.214,Y -551.979,Z 727.453,A 0.000,B 0.000,C 90.000,E1 117.513} C_DIS
LIN {X 0.114,Y -555.664,Z 727.447,A 0.000,B 0.000,C 90.000,E1 116.360} C_DIS
LIN {X -0.034,Y -558.111,Z 727.442,A 0.000,B 0.000,C 90.000,E1 115.540} C_DIS
LIN {X -0.155,Y -560.198,Z 727.437,A 0.000,B 0.000,C 90.000,E1 114.719} C_DIS
LIN {X -0.253,Y -562.059,Z 727.433,A 0.000,B 0.000,C 90.000,E1 113.898} C_DIS
LIN {X 0.182,Y -563.668,Z 727.428,A 0.000,B 0.000,C 90.000,E1 113.025} C_DIS
LIN {X 0.113,Y -565.028,Z 727.423,A 0.000,B 0.000,C 90.000,E1 112.206} C_DIS
LIN {X -0.022,Y -567.200,Z 727.416,A 0.000,B 0.000,C 90.000,E1 110.844} C_DIS
LIN {X 0.214,Y -569.281,Z 727.408,A 0.000,B 0.000,C 90.000,E1 109.450} C_DIS
LIN {X 0.116,Y -571.594,Z 727.399,A 0.000,B 0.000,C 90.000,E1 107.819} C_DIS
LIN {X -0.104,Y -573.779,Z 727.390,A 0.000,B 0.000,C 90.000,E1 106.205} C_DIS
LIN {X -0.082,Y -576.223,Z 727.379,A 0.000,B 0.000,C 90.000,E1 104.300} C_DIS
LIN {X -0.156,Y -578.550,Z 727.369,A 0.000,B 0.000,C 90.000,E1 102.411} C_DIS
LIN {X -0.302,Y -580.236,Z 727.361,A 0.000,B 0.000,C 90.000,E1 101.074} C_DIS
LIN {X 0.036,Y -581.603,Z 727.355,A 0.000,B 0.000,C 90.000,E1 99.962} C_DIS
LIN {X -0.286,Y -582.831,Z 727.349,A 0.000,B 0.000,C 90.000,E1 98.916} C_DIS
LIN {X 0.139,Y -584.255,Z 727.342,A 0.000,B 0.000,C 90.000,E1 97.530} C_DIS
LIN {X -0.163,Y -586.165,Z 727.332,A 0.000,B 0.000,C 90.000,E1 95.682} C_DIS
LIN {X -0.134,Y -587.707,Z 727.323,A 0.000,B 0.000,C 90.000,E1 94.073} C_DIS
LIN {X -0.074,Y -589.084,Z 727.314,A 0.000,B 0.000,C 90.000,E1 92.465} C_DIS
LIN {X -0.041,Y -589.671,Z 727.309,A 0.000,B 0.000,C 90.000,E1 91.661} C_DIS
LIN {X 0.007,Y -590.638,Z 727.300,A 0.000,B 0.000,C 90.000,E1 90.057} C_DIS
LIN {X 0.251,Y -591.182,Z 727.294,A 0.000,B 0.000,C 90.000,E1 88.969} C_DIS
LIN {X 0.133,Y -591.695,Z 727.287,A 0.000,B 0.000,C 90.000,E1 87.650} C_DIS
LIN {X -0.181,Y -591.990,Z 727.281,A 0.000,B 0.000,C 90.000,E1 86.617} C_DIS
LIN {X -0.036,Y -592.280,Z 727.272,A 0.000,B 0.000,C 90.000,E1 85.008} C_DIS
LIN {X 0.296,Y -592.387,Z 727.266,A 0.000,B 0.000,C 90.000,E1 83.913} C_DIS
LIN {X -0.089,Y -592.401,Z 727.258,A 0.000,B 0.000,C 90.000,E1 82.356} C_DIS
LIN {X -0.085,Y -592.205,Z 727.250,A 0.000,B 0.000,C 90.000,E1 81.027} C_DIS
LIN {X 0.002,Y -591.831,Z 727.243,A 0.000,B 0.000,C 90.000,E1 79.690} C_DIS
LIN {X 0.198,Y -591.156,Z 727.235,A 0.000,B 0.000,C 90.000,E1 78.342} C_DIS
LIN {X 0.078,Y -590.277,Z 727.227,A 0.000,B 0.000,C 90.000,E1 76.756} C_DIS
LIN {X -0.073,Y -589.219,Z 727.218,A 0.000,B 0.000,C 90.000,E1 75.172} C_DIS
LIN {X -0.196,Y -588.160,Z 727.210,A 0.000,B 0.000,C 90.000,E1 73.850} C_DIS
LIN {X -0.175,Y -587.312,Z 727.204,A 0.000,B 0.000,C 90.000,E1 72.779} C_DIS
LIN {X 0.006,Y -586.337,Z 727.198,A 0.000,B 0.000,C 90.000,E1 71.692} C_DIS
LIN {X 0.249,Y -584.693,Z 727.189,A 0.000,B 0.000,C 90.000,E1 70.061} C_DIS
LIN {X 0.240,Y -583.091,Z 727.182,A 0.000,B 0.000,C 90.000,E1 68.720} C_DIS
LIN {X -0.124,Y -581.400,Z 727.174,A 0.000,B 0.000,C 90.000,E1 67.411} C_DIS
LIN {X 0.161,Y -579.802,Z 727.169,A 0.000,B 0.000,C 90.000,E1 66.305} C_DIS
LIN {X 0.121,Y -578.031,Z 727.162,A 0.000,B 0.000,C 90.000,E1 65.229} C_DIS
LIN {X 0.058,Y -576.017,Z 727.156,A 0.000,B 0.000,C 90.000,E1 64.152} C_DIS
LIN {X -0.036,Y -573.685,Z 727.150,A 0.000,B 0.000,C 90.000,E1 63.076} C_DIS
LIN {X -0.089,Y -572.480,Z 727.147,A 0.000,B 0.000,C 90.000,E1 62.538} C_DIS
LIN {X 0.029,Y -569.625,Z 727.141,A 0.000,B 0.000,C 90.000,E1 61.435} C_DIS
LIN {X 0.284,Y -567.328,Z 727.137,A 0.000,B 0.000,C 90.000,E1 60.589} C_DIS
LIN {X 0.017,Y -564.860,Z 727.132,A 0.000,B 0.000,C 90.000,E1 59.793} C_DIS
LIN {X -0.272,Y -562.121,Z 727.128,A 0.000,B 0.000,C 90.000,E1 58.997} C_DIS
LIN {X 0.179,Y -559.178,Z 727.123,A 0.000,B 0.000,C 90.000,E1 58.122} C_DIS
LIN {X 0.047,Y -557.064,Z 727.120,A 0.000,B 0.000,C 90.000,E1 57.582} C_DIS
LIN {X -0.027,Y -553.557,Z 727.115,A 0.000,B 0.000,C 90.000,E1 56.755} C_DIS
LIN {X -0.323,Y -550.225,Z 727.111,A 0.000,B 0.000,C 90.000,E1 56.087} C_DIS
LIN {X -0.311,Y -546.654,Z 727.108,A 0.000,B 0.000,C 90.000,E1 55.388} C_DIS
LIN {X 0.079,Y -542.608,Z 727.104,A 0.000,B 0.000,C 90.000,E1 54.642} C_DIS
LIN {X 0.152,Y -539.258,Z 727.101,A 0.000,B 0.000,C 90.000,E1 54.069} C_DIS
LIN {X 0.183,Y -535.570,Z 727.097,A 0.000,B 0.000,C 90.000,E1 53.497} C_DIS
LIN {X 0.186,Y -531.477,Z 727.094,A 0.000,B 0.000,C 90.000,E1 52.924} C_DIS
LIN {X 0.160,Y -527.016,Z 727.091,A 0.000,B 0.000,C 90.000,E1 52.351} C_DIS
LIN {X -0.273,Y -521.850,Z 727.088,A 0.000,B 0.000,C 90.000,E1 51.823} C_DIS
LIN {X 0.085,Y -518.328,Z 727.086,A 0.000,B 0.000,C 90.000,E1 51.412} C_DIS
LIN {X -0.128,Y -512.813,Z 727.083,A 0.000,B 0.000,C 90.000,E1 50.928} C_DIS
LIN {X -0.251,Y -506.777,Z 727.080,A 0.000,B 0.000,C 90.000,E1 50.436} C_DIS
LIN {X -0.228,Y -502.136,Z 727.078,A 0.000,B 0.000,C 90.000,E1 50.070} C_DIS
LIN {X 0.068,Y -495.710,Z 727.076,A 0.000,B 0.000,C 90.000,E1 49.585} C_DIS
LIN {X -0.065,Y -489.135,Z 727.073,A 0.000,B 0.000,C 90.000,E1 49.175} C_DIS
LIN {X 0.246,Y -476.012,Z 727.069,A 0.000,B 0.000,C 90.000,E1 48.324} C_DIS
LIN {X -0.164,Y -454.936,Z 727.061,A 0.000,B 0.000,C 90.000,E1 47.067} C_DIS
LIN {X -0.046,Y -424.101,Z 727.050,A 0.000,B 0.000,C 90.000,E1 45.000} C_DIS
LIN {X -0.165,Y -417.869,Z 727.047,A 0.000,B 0.000,C 90.000,E1 44.514} C_DIS
LIN {X -0.194,Y -417.831,Z 727.047,A 0.000,B 0.000,C 90.000,E1 44.514} C_DIS
LIN {X -0.208,Y -408.362,Z 727.022,A 0.000,B 0.000,C 90.000,E1 40.011} C_DIS
LIN {X 0.073,Y -406.049,Z 727.014,A 0.000,B 0.000,C 90.000,E1 38.588} C_DIS
LIN {X -0.079,Y -405.199,Z 727.012,A 0.000,B 0.000,C 90.000,E1 38.177} C_DIS
LIN {X 0.152,Y -405.638,Z 726.995,A 0.000,B 0.000,C 90.000,E1 35.105} C_DIS
LIN {X -0.016,Y -406.828,Z 726.978,A 0.000,B 0.000,C 90.000,E1 32.005} C_DIS
LIN {X 0.017,Y -407.770,Z 726.966,A 0.000,B 0.000,C 90.000,E1 29.922} C_DIS
LIN {X 0.025,Y -408.953,Z 726.955,A 0.000,B 0.000,C 90.000,E1 27.847} C_DIS
LIN {X 0.165,Y -410.439,Z 726.941,A 0.000,B 0.000,C 90.000,E1 25.412} C_DIS
LIN {X -0.093,Y -412.628,Z 726.926,A 0.000,B 0.000,C 90.000,E1 22.695} C_DIS
LIN {X -0.037,Y -414.208,Z 726.917,A 0.000,B 0.000,C 90.000,E1 20.972} C_DIS
LIN {X 0.058,Y -416.329,Z 726.905,A 0.000,B 0.000,C 90.000,E1 18.906} C_DIS
LIN {X 0.239,Y -419.224,Z 726.892,A 0.000,B 0.000,C 90.000,E1 16.496} C_DIS
LIN {X -0.080,Y -422.902,Z 726.877,A 0.000,B 0.000,C 90.000,E1 13.828} C_DIS
LIN {X 0.171,Y -425.770,Z 726.866,A 0.000,B 0.000,C 90.000,E1 11.771} C_DIS
LIN {X -0.195,Y -428.273,Z 726.856,A 0.000,B 0.000,C 90.000,E1 10.141} C_DIS
LIN {X 0.134,Y -431.780,Z 726.843,A 0.000,B 0.000,C 90.000,E1 7.757} C_DIS
LIN {X -0.041,Y -435.246,Z 726.830,A 0.000,B 0.000,C 90.000,E1 5.454} C_DIS
LIN {X -0.021,Y -439.613,Z 726.816,A 0.000,B 0.000,C 90.000,E1 2.808} C_DIS
LIN {X 0.067,Y -444.255,Z 726.801,A 0.000,B 0.000,C 90.000,E1 0.172} C_DIS
LIN {X -0.012,Y -448.206,Z 726.790,A 0.000,B 0.000,C 90.000,E1 358.165} C_DIS
LIN {X 0.085,Y -454.132,Z 726.774,A 0.000,B 0.000,C 90.000,E1 355.241} C_DIS
LIN {X 0.140,Y -457.611,Z 726.765,A 0.000,B 0.000,C 90.000,E1 353.628} C_DIS
LIN {X -0.133,Y -460.999,Z 726.756,A 0.000,B 0.000,C 90.000,E1 352.064} C_DIS
LIN {X 0.177,Y -465.573,Z 726.744,A 0.000,B 0.000,C 90.000,E1 349.803} C_DIS
LIN {X -0.137,Y -468.047,Z 726.737,A 0.000,B 0.000,C 90.000,E1 348.578} C_DIS
LIN {X -0.218,Y -471.502,Z 726.726,A 0.000,B 0.000,C 90.000,E1 346.700} C_DIS
LIN {X 0.058,Y -474.356,Z 726.717,A 0.000,B 0.000,C 90.000,E1 345.102} C_DIS
LIN {X 0.192,Y -478.441,Z 726.705,A 0.000,B 0.000,C 90.000,E1 342.906} C_DIS
LIN {X -0.187,Y -481.744,Z 726.697,A 0.000,B 0.000,C 90.000,E1 341.402} C_DIS
LIN {X -0.198,Y -483.384,Z 726.693,A 0.000,B 0.000,C 90.000,E1 340.786} C_DIS
LIN {X 0.034,Y -484.814,Z 726.691,A 0.000,B 0.000,C 90.000,E1 340.296} C_DIS
LIN {X 0.229,Y -486.996,Z 726.688,A 0.000,B 0.000,C 90.000,E1 339.752} C_DIS
LIN {X 0.074,Y -488.658,Z 726.686,A 0.000,B 0.000,C 90.000,E1 339.464} C_DIS
LIN {X 0.068,Y -492.209,Z 726.683,A 0.000,B 0.000,C 90.000,E1 338.954} C_DIS
LIN {X 0.155,Y -494.932,Z 726.682,A 0.000,B 0.000,C 90.000,E1 338.646} C_DIS
LIN {X -0.008,Y -498.616,Z 726.680,A 0.000,B 0.000,C 90.000,E1 338.337} C_DIS
LIN {X -0.066,Y -504.389,Z 726.677,A 0.000,B 0.000,C 90.000,E1 337.901} C_DIS
LIN {X 0.310,Y -529.838,Z 726.668,A 0.000,B 0.000,C 90.000,E1 336.230} C_DIS
LIN {X -0.246,Y -537.557,Z 726.665,A 0.000,B 0.000,C 90.000,E1 335.793} C_DIS
LIN {X -0.238,Y -541.962,Z 726.664,A 0.000,B 0.000,C 90.000,E1 335.485} C_DIS
LIN {X 0.264,Y -546.385,Z 726.662,A 0.000,B 0.000,C 90.000,E1 335.101} C_DIS
LIN {X -0.015,Y -552.000,Z 726.659,A 0.000,B 0.000,C 90.000,E1 334.665} C_DIS
LIN {X 0.230,Y -557.451,Z 726.657,A 0.000,B 0.000,C 90.000,E1 334.152} C_DIS
LIN {X -0.129,Y -563.980,Z 726.653,A 0.000,B 0.000,C 90.000,E1 333.563} C_DIS
LIN {X 0.300,Y -569.111,Z 726.650,A 0.000,B 0.000,C 90.000,E1 332.999} C_DIS
LIN {X 0.079,Y -574.074,Z 726.647,A 0.000,B 0.000,C 90.000,E1 332.487} C_DIS
LIN {X 0.279,Y -583.763,Z 726.641,A 0.000,B 0.000,C 90.000,E1 331.385} C_DIS
LIN {X 0.249,Y -589.354,Z 726.638,A 0.000,B 0.000,C 90.000,E1 330.717} C_DIS
LIN {X 0.174,Y -596.834,Z 726.632,A 0.000,B 0.000,C 90.000,E1 329.793} C_DIS
LIN {X 0.223,Y -602.955,Z 726.628,A 0.000,B 0.000,C 90.000,E1 328.997} C_DIS
LIN {X -0.212,Y -609.799,Z 726.623,A 0.000,B 0.000,C 90.000,E1 328.122} C_DIS
LIN {X -0.038,Y -615.292,Z 726.619,A 0.000,B 0.000,C 90.000,E1 327.327} C_DIS
LIN {X -0.006,Y -621.340,Z 726.614,A 0.000,B 0.000,C 90.000,E1 326.421} C_DIS
LIN {X -0.241,Y -626.149,Z 726.609,A 0.000,B 0.000,C 90.000,E1 325.674} C_DIS
LIN {X 0.286,Y -632.278,Z 726.604,A 0.000,B 0.000,C 90.000,E1 324.609} C_DIS
LIN {X 0.148,Y -636.577,Z 726.599,A 0.000,B 0.000,C 90.000,E1 323.863} C_DIS
LIN {X -0.193,Y -642.656,Z 726.593,A 0.000,B 0.000,C 90.000,E1 322.763} C_DIS
LIN {X 0.144,Y -646.507,Z 726.589,A 0.000,B 0.000,C 90.000,E1 321.984} C_DIS
LIN {X -0.049,Y -651.970,Z 726.583,A 0.000,B 0.000,C 90.000,E1 320.884} C_DIS
LIN {X -0.190,Y -656.508,Z 726.577,A 0.000,B 0.000,C 90.000,E1 319.908} C_DIS
LIN {X -0.274,Y -660.737,Z 726.572,A 0.000,B 0.000,C 90.000,E1 318.933} C_DIS
LIN {X 0.135,Y -664.737,Z 726.566,A 0.000,B 0.000,C 90.000,E1 317.919} C_DIS
LIN {X 0.150,Y -668.364,Z 726.561,A 0.000,B 0.000,C 90.000,E1 316.944} C_DIS
LIN {X 0.178,Y -671.785,Z 726.556,A 0.000,B 0.000,C 90.000,E1 315.972} C_DIS
LIN {X 0.255,Y -675.005,Z 726.550,A 0.000,B 0.000,C 90.000,E1 315.000} C_DIS
LIN {X 0.342,Y -677.291,Z 726.546,A 0.000,B 0.000,C 90.000,E1 314.271} C_DIS
LIN {X 0.064,Y -680.841,Z 726.539,A 0.000,B 0.000,C 90.000,E1 313.095} C_DIS
LIN {X -0.161,Y -684.146,Z 726.533,A 0.000,B 0.000,C 90.000,E1 311.919} C_DIS
LIN {X -0.004,Y -685.998,Z 726.529,A 0.000,B 0.000,C 90.000,E1 311.191} C_DIS
LIN {X -0.094,Y -688.779,Z 726.522,A 0.000,B 0.000,C 90.000,E1 310.011} C_DIS
LIN {X 0.241,Y -690.648,Z 726.517,A 0.000,B 0.000,C 90.000,E1 309.036} C_DIS
LIN {X 0.166,Y -692.287,Z 726.512,A 0.000,B 0.000,C 90.000,E1 308.096} C_DIS
LIN {X 0.114,Y -693.686,Z 726.507,A 0.000,B 0.000,C 90.000,E1 307.156} C_DIS
LIN {X 0.078,Y -694.919,Z 726.501,A 0.000,B 0.000,C 90.000,E1 306.217} C_DIS
LIN {X -0.354,Y -696.003,Z 726.496,A 0.000,B 0.000,C 90.000,E1 305.311} C_DIS
LIN {X -0.146,Y -697.101,Z 726.490,A 0.000,B 0.000,C 90.000,E1 304.119} C_DIS
LIN {X -0.031,Y -698.480,Z 726.480,A 0.000,B 0.000,C 90.000,E1 302.467} C_DIS
LIN {X 0.073,Y -699.638,Z 726.473,A 0.000,B 0.000,C 90.000,E1 301.052} C_DIS
LIN {X 0.257,Y -700.127,Z 726.469,A 0.000,B 0.000,C 90.000,E1 300.335} C_DIS
LIN {X 0.039,Y -700.494,Z 726.461,A 0.000,B 0.000,C 90.000,E1 298.949} C_DIS
LIN {X 0.163,Y -700.839,Z 726.454,A 0.000,B 0.000,C 90.000,E1 297.769} C_DIS
LIN {X 0.134,Y -701.695,Z 726.443,A 0.000,B 0.000,C 90.000,E1 295.668} C_DIS
LIN {X 0.054,Y -701.881,Z 726.440,A 0.000,B 0.000,C 90.000,E1 295.207} C_DIS
LIN {X -0.326,Y -701.760,Z 726.438,A 0.000,B 0.000,C 90.000,E1 294.771} C_DIS
LIN {X -0.050,Y -701.590,Z 726.436,A 0.000,B 0.000,C 90.000,E1 294.515} C_DIS
LIN {X 0.211,Y -700.127,Z 726.434,A 0.000,B 0.000,C 90.000,E1 294.027} C_DIS
LIN {X -0.157,Y -699.179,Z 726.432,A 0.000,B 0.000,C 90.000,E1 293.823} C_DIS
LIN {X -0.025,Y -698.304,Z 726.432,A 0.000,B 0.000,C 90.000,E1 293.695} C_DIS
LIN {X 0.109,Y -697.090,Z 726.431,A 0.000,B 0.000,C 90.000,E1 293.567} C_DIS
LIN {X -0.241,Y -692.999,Z 726.429,A 0.000,B 0.000,C 90.000,E1 293.259} C_DIS
LIN {X 0.017,Y -691.501,Z 726.429,A 0.000,B 0.000,C 90.000,E1 293.131} C_DIS
LIN {X 0.088,Y -689.262,Z 726.428,A 0.000,B 0.000,C 90.000,E1 293.025} C_DIS
LIN {X -0.204,Y -686.586,Z 726.427,A 0.000,B 0.000,C 90.000,E1 292.950} C_DIS
LIN {X -0.105,Y -680.559,Z 726.427,A 0.000,B 0.000,C 90.000,E1 292.770} C_DIS
LIN {X 0.346,Y -676.750,Z 726.426,A 0.000,B 0.000,C 90.000,E1 292.642} C_DIS
LIN {X -0.195,Y -658.880,Z 726.425,A 0.000,B 0.000,C 90.000,E1 292.461} C_DIS
LIN {X 0.084,Y -648.543,Z 726.424,A 0.000,B 0.000,C 90.000,E1 292.280} C_DIS
LIN {X 0.294,Y -638.645,Z 726.423,A 0.000,B 0.000,C 90.000,E1 292.078} C_DIS
LIN {X -0.075,Y -628.754,Z 726.422,A 0.000,B 0.000,C 90.000,E1 291.897} C_DIS
LIN {X 0.002,Y -611.693,Z 726.419,A 0.000,B 0.000,C 90.000,E1 291.461} C_DIS
LIN {X 0.085,Y -580.413,Z 726.414,A 0.000,B 0.000,C 90.000,E1 290.556} C_DIS
LIN {X -0.346,Y -567.752,Z 726.412,A 0.000,B 0.000,C 90.000,E1 290.248} C_DIS
LIN {X -0.072,Y -561.139,Z 726.411,A 0.000,B 0.000,C 90.000,E1 289.993} C_DIS
LIN {X -0.036,Y -558.976,Z 726.410,A 0.000,B 0.000,C 90.000,E1 289.866} C_DIS
LIN {X 0.032,Y -556.555,Z 726.410,A 0.000,B 0.000,C 90.000,E1 289.704} C_DIS
LIN {X 0.002,Y -556.508,Z 726.410,A 0.000,B 0.000,C 90.000,E1 289.704} C_DIS
LIN {X 0.020,Y -555.512,Z 726.409,A 0.000,B 0.000,C 90.000,E1 289.523} C_DIS
LIN {X 0.191,Y -554.857,Z 726.406,A 0.000,B 0.000,C 90.000,E1 289.087} C_DIS
LIN {X 0.103,Y -554.509,Z 726.400,A 0.000,B 0.000,C 90.000,E1 288.055} C_DIS
LIN {X -0.216,Y -553.738,Z 726.390,A 0.000,B 0.000,C 90.000,E1 286.134} C_DIS
LIN {X -0.178,Y -553.047,Z 726.379,A 0.000,B 0.000,C 90.000,E1 284.175} C_DIS
LIN {X 0.123,Y -552.437,Z 726.368,A 0.000,B 0.000,C 90.000,E1 282.187} C_DIS
LIN {X -0.122,Y -551.639,Z 726.357,A 0.000,B 0.000,C 90.000,E1 280.254} C_DIS
LIN {X -0.181,Y -550.993,Z 726.349,A 0.000,B 0.000,C 90.000,E1 278.859} C_DIS
LIN {X -0.120,Y -550.059,Z 726.338,A 0.000,B 0.000,C 90.000,E1 276.891} C_DIS
LIN {X -0.209,Y -549.362,Z 726.327,A 0.000,B 0.000,C 90.000,E1 274.935} C_DIS
LIN {X 0.105,Y -548.837,Z 726.320,A 0.000,B 0.000,C 90.000,E1 273.498} C_DIS
LIN {X -0.058,Y -548.020,Z 726.309,A 0.000,B 0.000,C 90.000,E1 271.547} C_DIS
LIN {X 0.133,Y -547.428,Z 726.302,A 0.000,B 0.000,C 90.000,E1 270.401} C_DIS
LIN {X -0.142,Y -546.393,Z 726.293,A 0.000,B 0.000,C 90.000,E1 268.740} C_DIS
LIN {X 0.114,Y -545.332,Z 726.284,A 0.000,B 0.000,C 90.000,E1 267.020} C_DIS
LIN {X -0.229,Y -544.587,Z 726.277,A 0.000,B 0.000,C 90.000,E1 265.927} C_DIS
LIN {X 0.020,Y -543.396,Z 726.268,A 0.000,B 0.000,C 90.000,E1 264.204} C_DIS
LIN {X 0.272,Y -542.320,Z 726.260,A 0.000,B 0.000,C 90.000,E1 262.761} C_DIS
LIN {X 0.038,Y -540.872,Z 726.251,A 0.000,B 0.000,C 90.000,E1 261.084} C_DIS
LIN {X -0.288,Y -539.910,Z 726.244,A 0.000,B 0.000,C 90.000,E1 259.982} C_DIS
LIN {X -0.255,Y -537.981,Z 726.232,A 0.000,B 0.000,C 90.000,E1 257.701} C_DIS
LIN {X 0.186,Y -536.745,Z 726.224,A 0.000,B 0.000,C 90.000,E1 256.228} C_DIS
LIN {X 0.028,Y -535.654,Z 726.217,A 0.000,B 0.000,C 90.000,E1 255.102} C_DIS
LIN {X 0.090,Y -533.836,Z 726.208,A 0.000,B 0.000,C 90.000,E1 253.378} C_DIS
LIN {X 0.260,Y -532.089,Z 726.198,A 0.000,B 0.000,C 90.000,E1 251.638} C_DIS
LIN {X 0.161,Y -531.112,Z 726.193,A 0.000,B 0.000,C 90.000,E1 250.786} C_DIS
LIN {X 0.058,Y -529.546,Z 726.187,A 0.000,B 0.000,C 90.000,E1 249.645} C_DIS
LIN {X 0.300,Y -528.012,Z 726.181,A 0.000,B 0.000,C 90.000,E1 248.465} C_DIS
LIN {X -0.161,Y -526.335,Z 726.174,A 0.000,B 0.000,C 90.000,E1 247.358} C_DIS
LIN {X 0.038,Y -524.616,Z 726.168,A 0.000,B 0.000,C 90.000,E1 246.177} C_DIS
LIN {X -0.049,Y -522.747,Z 726.161,A 0.000,B 0.000,C 90.000,E1 245.025} C_DIS
LIN {X 0.086,Y -520.874,Z 726.155,A 0.000,B 0.000,C 90.000,E1 243.845} C_DIS
LIN {X -0.146,Y -518.208,Z 726.147,A 0.000,B 0.000,C 90.000,E1 242.410} C_DIS
LIN {X 0.038,Y -515.344,Z 726.139,A 0.000,B 0.000,C 90.000,E1 240.923} C_DIS
LIN {X -0.032,Y -512.398,Z 726.130,A 0.000,B 0.000,C 90.000,E1 239.459} C_DIS
LIN {X -0.155,Y -509.385,Z 726.122,A 0.000,B 0.000,C 90.000,E1 237.995} C_DIS
LIN {X -0.069,Y -506.246,Z 726.114,A 0.000,B 0.000,C 90.000,E1 236.501} C_DIS
LIN {X 0.233,Y -503.037,Z 726.106,A 0.000,B 0.000,C 90.000,E1 234.975} C_DIS
LIN {X 0.181,Y -500.136,Z 726.099,A 0.000,B 0.000,C 90.000,E1 233.783} C_DIS
LIN {X -0.013,Y -497.156,Z 726.092,A 0.000,B 0.000,C 90.000,E1 232.603} C_DIS
LIN {X 0.007,Y -493.275,Z 726.084,A 0.000,B 0.000,C 90.000,E1 231.090} C_DIS
LIN {X -0.118,Y -489.635,Z 726.075,A 0.000,B 0.000,C 90.000,E1 229.585} C_DIS
LIN {X 0.052,Y -486.200,Z 726.067,A 0.000,B 0.000,C 90.000,E1 228.038} C_DIS
LIN {X -0.113,Y -481.984,Z 726.057,A 0.000,B 0.000,C 90.000,E1 226.215} C_DIS
LIN {X -0.149,Y -478.563,Z 726.048,A 0.000,B 0.000,C 90.000,E1 224.676} C_DIS
LIN {X 0.094,Y -475.303,Z 726.040,A 0.000,B 0.000,C 90.000,E1 223.095} C_DIS
LIN {X 0.044,Y -471.343,Z 726.029,A 0.000,B 0.000,C 90.000,E1 221.229} C_DIS
LIN {X -0.251,Y -468.651,Z 726.022,A 0.000,B 0.000,C 90.000,E1 220.011} C_DIS
LIN {X 0.187,Y -465.094,Z 726.013,A 0.000,B 0.000,C 90.000,E1 218.382} C_DIS
LIN {X -0.013,Y -461.602,Z 726.005,A 0.000,B 0.000,C 90.000,E1 216.824} C_DIS
LIN {X 0.111,Y -457.675,Z 725.994,A 0.000,B 0.000,C 90.000,E1 214.898} C_DIS
LIN {X -0.035,Y -453.394,Z 725.982,A 0.000,B 0.000,C 90.000,E1 212.673} C_DIS
LIN {X -0.016,Y -449.251,Z 725.969,A 0.000,B 0.000,C 90.000,E1 210.413} C_DIS
LIN {X -0.242,Y -446.184,Z 725.960,A 0.000,B 0.000,C 90.000,E1 208.821} C_DIS
LIN {X -0.200,Y -443.781,Z 725.953,A 0.000,B 0.000,C 90.000,E1 207.513} C_DIS
LIN {X -0.006,Y -441.423,Z 725.945,A 0.000,B 0.000,C 90.000,E1 206.181} C_DIS
LIN {X -0.140,Y -437.184,Z 725.933,A 0.000,B 0.000,C 90.000,E1 203.898} C_DIS
LIN {X -0.226,Y -434.758,Z 725.925,A 0.000,B 0.000,C 90.000,E1 202.589} C_DIS
LIN {X 0.050,Y -432.243,Z 725.918,A 0.000,B 0.000,C 90.000,E1 201.227} C_DIS
LIN {X -0.091,Y -430.473,Z 725.912,A 0.000,B 0.000,C 90.000,E1 200.248} C_DIS
LIN {X 0.166,Y -426.187,Z 725.899,A 0.000,B 0.000,C 90.000,E1 197.873} C_DIS
LIN {X 0.071,Y -422.943,Z 725.890,A 0.000,B 0.000,C 90.000,E1 196.205} C_DIS
LIN {X 0.140,Y -418.678,Z 725.877,A 0.000,B 0.000,C 90.000,E1 193.828} C_DIS
LIN {X -0.160,Y -415.056,Z 725.866,A 0.000,B 0.000,C 90.000,E1 191.827} C_DIS
LIN {X -0.166,Y -410.270,Z 725.850,A 0.000,B 0.000,C 90.000,E1 189.086} C_DIS
LIN {X -0.119,Y -406.380,Z 725.837,A 0.000,B 0.000,C 90.000,E1 186.663} C_DIS
LIN {X 0.189,Y -402.757,Z 725.823,A 0.000,B 0.000,C 90.000,E1 184.188} C_DIS
LIN {X -0.046,Y -399.471,Z 725.810,A 0.000,B 0.000,C 90.000,E1 181.776} C_DIS
LIN {X -0.133,Y -395.881,Z 725.792,A 0.000,B 0.000,C 90.000,E1 178.625} C_DIS
LIN {X -0.178,Y -393.564,Z 725.779,A 0.000,B 0.000,C 90.000,E1 176.159} C_DIS
LIN {X 0.110,Y -391.361,Z 725.763,A 0.000,B 0.000,C 90.000,E1 173.280} C_DIS
LIN {X 0.221,Y -389.048,Z 725.737,A 0.000,B 0.000,C 90.000,E1 168.634} C_DIS
LIN {X -0.036,Y -388.140,Z 725.723,A 0.000,B 0.000,C 90.000,E1 166.172} C_DIS
LIN {X -0.082,Y -387.424,Z 725.705,A 0.000,B 0.000,C 90.000,E1 162.960} C_DIS
LIN {X 0.041,Y -387.229,Z 725.697,A 0.000,B 0.000,C 90.000,E1 161.511} C_DIS
LIN {X -0.148,Y -387.031,Z 725.685,A 0.000,B 0.000,C 90.000,E1 159.390} C_DIS
LIN {X -0.052,Y -386.843,Z 725.672,A 0.000,B 0.000,C 90.000,E1 156.869} C_DIS
LIN {X 0.144,Y -386.934,Z 725.662,A 0.000,B 0.000,C 90.000,E1 155.049} C_DIS
LIN {X -0.007,Y -387.173,Z 725.648,A 0.000,B 0.000,C 90.000,E1 152.564} C_DIS
LIN {X 0.026,Y -387.658,Z 725.636,A 0.000,B 0.000,C 90.000,E1 150.411} C_DIS
LIN {X 0.082,Y -392.157,Z 725.598,A 0.000,B 0.000,C 90.000,E1 143.623} C_DIS
LIN {X 0.163,Y -396.735,Z 725.578,A 0.000,B 0.000,C 90.000,E1 140.070} C_DIS
LIN {X 0.159,Y -398.628,Z 725.572,A 0.000,B 0.000,C 90.000,E1 139.013} C_DIS
LIN {X 0.069,Y -400.391,Z 725.569,A 0.000,B 0.000,C 90.000,E1 138.324} C_DIS
LIN {X -0.009,Y -402.656,Z 725.565,A 0.000,B 0.000,C 90.000,E1 137.634} C_DIS
LIN {X -0.100,Y -403.334,Z 725.564,A 0.000,B 0.000,C 90.000,E1 137.472} C_DIS
LIN {X 0.019,Y -405.074,Z 725.562,A 0.000,B 0.000,C 90.000,E1 137.106} C_DIS
LIN {X -0.069,Y -405.878,Z 725.561,A 0.000,B 0.000,C 90.000,E1 136.944} C_DIS
LIN {X -0.036,Y -409.496,Z 725.558,A 0.000,B 0.000,C 90.000,E1 136.419} C_DIS
LIN {X 0.252,Y -415.264,Z 725.554,A 0.000,B 0.000,C 90.000,E1 135.729} C_DIS
LIN {X -0.170,Y -438.887,Z 725.541,A 0.000,B 0.000,C 90.000,E1 133.461} C_DIS
LIN {X -0.136,Y -450.695,Z 725.535,A 0.000,B 0.000,C 90.000,E1 132.366} C_DIS
LIN {X -0.067,Y -458.078,Z 725.532,A 0.000,B 0.000,C 90.000,E1 131.676} C_DIS
LIN {X -0.045,Y -465.295,Z 725.528,A 0.000,B 0.000,C 90.000,E1 130.987} C_DIS
LIN {X -0.092,Y -473.791,Z 725.523,A 0.000,B 0.000,C 90.000,E1 130.172} C_DIS
LIN {X 0.031,Y -479.336,Z 725.520,A 0.000,B 0.000,C 90.000,E1 129.600} C_DIS
LIN {X -0.006,Y -484.550,Z 725.517,A 0.000,B 0.000,C 90.000,E1 129.072} C_DIS
LIN {X -0.195,Y -491.255,Z 725.513,A 0.000,B 0.000,C 90.000,E1 128.382} C_DIS
LIN {X -0.323,Y -496.550,Z 725.510,A 0.000,B 0.000,C 90.000,E1 127.810} C_DIS
LIN {X 0.211,Y -501.515,Z 725.507,A 0.000,B 0.000,C 90.000,E1 127.156} C_DIS
LIN {X -0.011,Y -506.427,Z 725.503,A 0.000,B 0.000,C 90.000,E1 126.583} C_DIS
LIN {X -0.015,Y -509.890,Z 725.501,A 0.000,B 0.000,C 90.000,E1 126.137} C_DIS
LIN {X 0.221,Y -514.183,Z 725.497,A 0.000,B 0.000,C 90.000,E1 125.518} C_DIS
LIN {X 0.248,Y -522.496,Z 725.490,A 0.000,B 0.000,C 90.000,E1 124.199} C_DIS
LIN {X -0.012,Y -526.502,Z 725.486,A 0.000,B 0.000,C 90.000,E1 123.499} C_DIS
LIN {X 0.201,Y -530.177,Z 725.482,A 0.000,B 0.000,C 90.000,E1 122.752} C_DIS
LIN {X -0.151,Y -534.219,Z 725.477,A 0.000,B 0.000,C 90.000,E1 121.926} C_DIS
LIN {X -0.002,Y -536.782,Z 725.474,A 0.000,B 0.000,C 90.000,E1 121.337} C_DIS
LIN {X 0.171,Y -540.344,Z 725.469,A 0.000,B 0.000,C 90.000,E1 120.463} C_DIS
LIN {X -0.145,Y -546.093,Z 725.461,A 0.000,B 0.000,C 90.000,E1 119.077} C_DIS
LIN {X 0.096,Y -550.364,Z 725.455,A 0.000,B 0.000,C 90.000,E1 117.924} C_DIS
LIN {X -0.119,Y -552.361,Z 725.452,A 0.000,B 0.000,C 90.000,E1 117.385} C_DIS
LIN {X -0.058,Y -555.189,Z 725.447,A 0.000,B 0.000,C 90.000,E1 116.539} C_DIS
LIN {X -0.217,Y -557.731,Z 725.443,A 0.000,B 0.000,C 90.000,E1 115.720} C_DIS
LIN {X -0.043,Y -560.579,Z 725.437,A 0.000,B 0.000,C 90.000,E1 114.591} C_DIS
LIN {X -0.139,Y -562.423,Z 725.432,A 0.000,B 0.000,C 90.000,E1 113.770} C_DIS
LIN {X -0.021,Y -563.562,Z 725.429,A 0.000,B 0.000,C 90.000,E1 113.206} C_DIS
LIN {X 0.234,Y -565.415,Z 725.423,A 0.000,B 0.000,C 90.000,E1 112.078} C_DIS
LIN {X -0.097,Y -567.595,Z 725.415,A 0.000,B 0.000,C 90.000,E1 110.737} C_DIS
LIN {X 0.154,Y -569.665,Z 725.408,A 0.000,B 0.000,C 90.000,E1 109.341} C_DIS
LIN {X -0.099,Y -571.651,Z 725.400,A 0.000,B 0.000,C 90.000,E1 108.000} C_DIS
LIN {X -0.155,Y -573.867,Z 725.391,A 0.000,B 0.000,C 90.000,E1 106.370} C_DIS
LIN {X 0.065,Y -575.967,Z 725.382,A 0.000,B 0.000,C 90.000,E1 104.717} C_DIS
LIN {X -0.084,Y -577.354,Z 725.376,A 0.000,B 0.000,C 90.000,E1 103.647} C_DIS
LIN {X -0.260,Y -579.776,Z 725.365,A 0.000,B 0.000,C 90.000,E1 101.771} C_DIS
LIN {X -0.148,Y -581.839,Z 725.356,A 0.000,B 0.000,C 90.000,E1 100.141} C_DIS
LIN {X 0.206,Y -583.109,Z 725.350,A 0.000,B 0.000,C 90.000,E1 99.029} C_DIS
LIN {X 0.053,Y -584.552,Z 725.343,A 0.000,B 0.000,C 90.000,E1 97.701} C_DIS
LIN {X -0.248,Y -586.489,Z 725.332,A 0.000,B 0.000,C 90.000,E1 95.853} C_DIS
LIN {X -0.218,Y -588.071,Z 725.323,A 0.000,B 0.000,C 90.000,E1 94.245} C_DIS
LIN {X 0.238,Y -589.239,Z 725.316,A 0.000,B 0.000,C 90.000,E1 92.865} C_DIS
LIN {X 0.087,Y -590.269,Z 725.309,A 0.000,B 0.000,C 90.000,E1 91.547} C_DIS
LIN {X -0.060,Y -591.089,Z 725.301,A 0.000,B 0.000,C 90.000,E1 90.229} C_DIS
LIN {X -0.191,Y -591.775,Z 725.294,A 0.000,B 0.000,C 90.000,E1 88.912} C_DIS
LIN {X -0.087,Y -592.358,Z 725.285,A 0.000,B 0.000,C 90.000,E1 87.306} C_DIS
LIN {X -0.188,Y -592.659,Z 725.278,A 0.000,B 0.000,C 90.000,E1 85.988} C_DIS
LIN {X -0.246,Y -592.851,Z 725.270,A 0.000,B 0.000,C 90.000,E1 84.666} C_DIS
LIN {X -0.113,Y -592.894,Z 725.266,A 0.000,B 0.000,C 90.000,E1 83.856} C_DIS
LIN {X -0.093,Y -592.911,Z 725.258,A 0.000,B 0.000,C 90.000,E1 82.527} C_DIS
LIN {X -0.074,Y -592.741,Z 725.251,A 0.000,B 0.000,C 90.000,E1 81.197} C_DIS
LIN {X 0.030,Y -592.371,Z 725.244,A 0.000,B 0.000,C 90.000,E1 79.859} C_DIS
LIN {X 0.159,Y -591.986,Z 725.239,A 0.000,B 0.000,C 90.000,E1 79.050} C_DIS
LIN {X 0.048,Y -591.095,Z 725.230,A 0.000,B 0.000,C 90.000,E1 77.465} C_DIS
LIN {X 0.229,Y -590.245,Z 725.223,A 0.000,B 0.000,C 90.000,E1 76.117} C_DIS
LIN {X -0.038,Y -589.315,Z 725.216,A 0.000,B 0.000,C 90.000,E1 74.810} C_DIS
LIN {X 0.093,Y -588.010,Z 725.207,A 0.000,B 0.000,C 90.000,E1 73.196} C_DIS
LIN {X 0.105,Y -587.036,Z 725.201,A 0.000,B 0.000,C 90.000,E1 72.127} C_DIS
LIN {X 0.136,Y -585.677,Z 725.193,A 0.000,B 0.000,C 90.000,E1 70.786} C_DIS
LIN {X -0.260,Y -584.555,Z 725.187,A 0.000,B 0.000,C 90.000,E1 69.752} C_DIS
LIN {X -0.269,Y -582.874,Z 725.180,A 0.000,B 0.000,C 90.000,E1 68.411} C_DIS
LIN {X 0.039,Y -581.447,Z 725.174,A 0.000,B 0.000,C 90.000,E1 67.305} C_DIS
LIN {X 0.157,Y -580.234,Z 725.169,A 0.000,B 0.000,C 90.000,E1 66.485} C_DIS
LIN {X 0.125,Y -578.449,Z 725.164,A 0.000,B 0.000,C 90.000,E1 65.409} C_DIS
LIN {X 0.218,Y -576.960,Z 725.159,A 0.000,B 0.000,C 90.000,E1 64.588} C_DIS
LIN {X 0.142,Y -574.709,Z 725.153,A 0.000,B 0.000,C 90.000,E1 63.512} C_DIS
LIN {X -0.323,Y -572.879,Z 725.148,A 0.000,B 0.000,C 90.000,E1 62.743} C_DIS
LIN {X -0.201,Y -570.066,Z 725.142,A 0.000,B 0.000,C 90.000,E1 61.641} C_DIS
LIN {X 0.056,Y -567.766,Z 725.138,A 0.000,B 0.000,C 90.000,E1 60.795} C_DIS
LIN {X -0.110,Y -564.375,Z 725.132,A 0.000,B 0.000,C 90.000,E1 59.715} C_DIS
LIN {X 0.080,Y -561.584,Z 725.127,A 0.000,B 0.000,C 90.000,E1 58.869} C_DIS
LIN {X -0.036,Y -559.635,Z 725.124,A 0.000,B 0.000,C 90.000,E1 58.329} C_DIS
LIN {X -0.085,Y -556.350,Z 725.119,A 0.000,B 0.000,C 90.000,E1 57.502} C_DIS
LIN {X 0.113,Y -553.390,Z 725.116,A 0.000,B 0.000,C 90.000,E1 56.786} C_DIS
LIN {X -0.012,Y -549.244,Z 725.111,A 0.000,B 0.000,C 90.000,E1 55.960} C_DIS
LIN {X 0.003,Y -545.511,Z 725.107,A 0.000,B 0.000,C 90.000,E1 55.261} C_DIS
LIN {X 0.079,Y -542.243,Z 725.104,A 0.000,B 0.000,C 90.000,E1 54.689} C_DIS
LIN {X 0.133,Y -538.795,Z 725.101,A 0.000,B 0.000,C 90.000,E1 54.116} C_DIS
LIN {X 0.163,Y -534.982,Z 725.098,A 0.000,B 0.000,C 90.000,E1 53.543} C_DIS
LIN {X -0.154,Y -530.826,Z 725.094,A 0.000,B 0.000,C 90.000,E1 53.004} C_DIS
LIN {X 0.139,Y -526.199,Z 725.091,A 0.000,B 0.000,C 90.000,E1 52.396} C_DIS
LIN {X 0.294,Y -521.138,Z 725.088,A 0.000,B 0.000,C 90.000,E1 51.823} C_DIS
LIN {X 0.165,Y -516.037,Z 725.085,A 0.000,B 0.000,C 90.000,E1 51.331} C_DIS
LIN {X -0.127,Y -511.508,Z 725.083,A 0.000,B 0.000,C 90.000,E1 50.964} C_DIS
LIN {X 0.212,Y -505.498,Z 725.080,A 0.000,B 0.000,C 90.000,E1 50.436} C_DIS
LIN {X -0.124,Y -500.718,Z 725.078,A 0.000,B 0.000,C 90.000,E1 50.114} C_DIS
LIN {X -0.017,Y -494.392,Z 725.076,A 0.000,B 0.000,C 90.000,E1 49.666} C_DIS
LIN {X 0.206,Y -487.840,Z 725.074,A 0.000,B 0.000,C 90.000,E1 49.218} C_DIS
LIN {X -0.042,Y -474.772,Z 725.069,A 0.000,B 0.000,C 90.000,E1 48.447} C_DIS
LIN {X -0.024,Y -451.861,Z 725.061,A 0.000,B 0.000,C 90.000,E1 47.025} C_DIS
LIN {X 0.202,Y -424.385,Z 725.051,A 0.000,B 0.000,C 90.000,E1 45.162} C_DIS
LIN {X 0.196,Y -418.370,Z 725.048,A 0.000,B 0.000,C 90.000,E1 44.676} C_DIS
LIN {X 0.170,Y -418.353,Z 725.048,A 0.000,B 0.000,C 90.000,E1 44.676} C_DIS
LIN {X 0.054,Y -408.716,Z 725.023,A 0.000,B 0.000,C 90.000,E1 40.172} C_DIS
LIN {X 0.146,Y -405.572,Z 725.013,A 0.000,B 0.000,C 90.000,E1 38.257} C_DIS
LIN {X 0.112,Y -405.989,Z 724.996,A 0.000,B 0.000,C 90.000,E1 35.311} C_DIS
LIN {X -0.042,Y -407.161,Z 724.979,A 0.000,B 0.000,C 90.000,E1 32.212} C_DIS
LIN {X -0.082,Y -408.303,Z 724.966,A 0.000,B 0.000,C 90.000,E1 29.795} C_DIS
LIN {X -0.061,Y -409.449,Z 724.954,A 0.000,B 0.000,C 90.000,E1 27.719} C_DIS
LIN {X 0.094,Y -410.975,Z 724.941,A 0.000,B 0.000,C 90.000,E1 25.283} C_DIS
LIN {X 0.231,Y -413.181,Z 724.925,A 0.000,B 0.000,C 90.000,E1 22.514} C_DIS
LIN {X 0.010,Y -414.449,Z 724.918,A 0.000,B 0.000,C 90.000,E1 21.173} C_DIS
LIN {X -0.133,Y -416.548,Z 724.906,A 0.000,B 0.000,C 90.000,E1 19.141} C_DIS
LIN {X 0.093,Y -419.815,Z 724.891,A 0.000,B 0.000,C 90.000,E1 16.386} C_DIS
LIN {X 0.071,Y -422.562,Z 724.880,A 0.000,B 0.000,C 90.000,E1 14.356} C_DIS
LIN {X -0.103,Y -425.391,Z 724.869,A 0.000,B 0.000,C 90.000,E1 12.355} C_DIS
LIN {X 0.117,Y -428.349,Z 724.857,A 0.000,B 0.000,C 90.000,E1 10.310} C_DIS
LIN {X 0.069,Y -432.267,Z 724.843,A 0.000,B 0.000,C 90.000,E1 7.644} C_DIS
LIN {X -0.047,Y -435.761,Z 724.830,A 0.000,B 0.000,C 90.000,E1 5.334} C_DIS
LIN {X -0.049,Y -440.075,Z 724.815,A 0.000,B 0.000,C 90.000,E1 2.694} C_DIS
LIN {X 0.000,Y -444.852,Z 724.800,A 0.000,B 0.000,C 90.000,E1 360.000} C_DIS
LIN {X -0.007,Y -448.455,Z 724.790,A 0.000,B 0.000,C 90.000,E1 358.165} C_DIS
LIN {X 0.099,Y -454.330,Z 724.774,A 0.000,B 0.000,C 90.000,E1 355.241} C_DIS
LIN {X 0.158,Y -457.809,Z 724.765,A 0.000,B 0.000,C 90.000,E1 353.628} C_DIS
LIN {X 0.064,Y -461.802,Z 724.754,A 0.000,B 0.000,C 90.000,E1 351.724} C_DIS
LIN {X -0.057,Y -465.103,Z 724.745,A 0.000,B 0.000,C 90.000,E1 350.151} C_DIS
LIN {X -0.108,Y -468.179,Z 724.737,A 0.000,B 0.000,C 90.000,E1 348.578} C_DIS
LIN {X -0.008,Y -471.068,Z 724.728,A 0.000,B 0.000,C 90.000,E1 346.992} C_DIS
LIN {X 0.093,Y -474.516,Z 724.717,A 0.000,B 0.000,C 90.000,E1 345.102} C_DIS
LIN {X -0.226,Y -478.567,Z 724.705,A 0.000,B 0.000,C 90.000,E1 342.960} C_DIS
LIN {X -0.153,Y -482.509,Z 724.695,A 0.000,B 0.000,C 90.000,E1 341.094} C_DIS
LIN {X 0.142,Y -485.110,Z 724.690,A 0.000,B 0.000,C 90.000,E1 340.134} C_DIS
LIN {X -0.074,Y -486.830,Z 724.687,A 0.000,B 0.000,C 90.000,E1 339.699} C_DIS
LIN {X 0.009,Y -489.551,Z 724.684,A 0.000,B 0.000,C 90.000,E1 339.156} C_DIS
LIN {X 0.033,Y -491.647,Z 724.683,A 0.000,B 0.000,C 90.000,E1 338.847} C_DIS
LIN {X -0.182,Y -492.850,Z 724.682,A 0.000,B 0.000,C 90.000,E1 338.720} C_DIS
LIN {X 0.096,Y -495.876,Z 724.680,A 0.000,B 0.000,C 90.000,E1 338.358} C_DIS
LIN {X 0.175,Y -501.138,Z 724.677,A 0.000,B 0.000,C 90.000,E1 337.922} C_DIS
LIN {X 0.105,Y -507.104,Z 724.675,A 0.000,B 0.000,C 90.000,E1 337.486} C_DIS
LIN {X 0.247,Y -529.340,Z 724.667,A 0.000,B 0.000,C 90.000,E1 336.049} C_DIS
LIN {X -0.138,Y -538.672,Z 724.664,A 0.000,B 0.000,C 90.000,E1 335.485} C_DIS
LIN {X -0.038,Y -544.577,Z 724.661,A 0.000,B 0.000,C 90.000,E1 335.049} C_DIS
LIN {X 0.052,Y -551.620,Z 724.658,A 0.000,B 0.000,C 90.000,E1 334.460} C_DIS
LIN {X 0.046,Y -557.165,Z 724.655,A 0.000,B 0.000,C 90.000,E1 333.973} C_DIS
LIN {X 0.095,Y -565.117,Z 724.651,A 0.000,B 0.000,C 90.000,E1 333.204} C_DIS
LIN {X 0.225,Y -571.429,Z 724.648,A 0.000,B 0.000,C 90.000,E1 332.538} C_DIS
LIN {X 0.041,Y -577.412,Z 724.644,A 0.000,B 0.000,C 90.000,E1 331.897} C_DIS
LIN {X -0.296,Y -583.408,Z 724.640,A 0.000,B 0.000,C 90.000,E1 331.257} C_DIS
LIN {X 0.184,Y -589.045,Z 724.636,A 0.000,B 0.000,C 90.000,E1 330.539} C_DIS
LIN {X 0.100,Y -596.650,Z 724.631,A 0.000,B 0.000,C 90.000,E1 329.616} C_DIS
LIN {X -0.102,Y -603.820,Z 724.626,A 0.000,B 0.000,C 90.000,E1 328.712} C_DIS
LIN {X -0.011,Y -610.629,Z 724.621,A 0.000,B 0.000,C 90.000,E1 327.788} C_DIS
LIN {X 0.192,Y -615.221,Z 724.617,A 0.000,B 0.000,C 90.000,E1 327.120} C_DIS
LIN {X -0.101,Y -620.452,Z 724.613,A 0.000,B 0.000,C 90.000,E1 326.373} C_DIS
LIN {X 0.003,Y -625.327,Z 724.609,A 0.000,B 0.000,C 90.000,E1 325.595} C_DIS
LIN {X 0.162,Y -630.740,Z 724.604,A 0.000,B 0.000,C 90.000,E1 324.689} C_DIS
LIN {X 0.380,Y -635.155,Z 724.600,A 0.000,B 0.000,C 90.000,E1 323.909} C_DIS
LIN {X -0.360,Y -641.336,Z 724.593,A 0.000,B 0.000,C 90.000,E1 322.844} C_DIS
LIN {X 0.368,Y -645.880,Z 724.589,A 0.000,B 0.000,C 90.000,E1 321.904} C_DIS
LIN {X -0.253,Y -650.824,Z 724.583,A 0.000,B 0.000,C 90.000,E1 320.964} C_DIS
LIN {X -0.367,Y -653.748,Z 724.580,A 0.000,B 0.000,C 90.000,E1 320.356} C_DIS
LIN {X 0.012,Y -658.229,Z 724.574,A 0.000,B 0.000,C 90.000,E1 319.337} C_DIS
LIN {X -0.112,Y -662.425,Z 724.569,A 0.000,B 0.000,C 90.000,E1 318.366} C_DIS
LIN {X -0.121,Y -666.250,Z 724.563,A 0.000,B 0.000,C 90.000,E1 317.391} C_DIS
LIN {X -0.126,Y -668.984,Z 724.559,A 0.000,B 0.000,C 90.000,E1 316.662} C_DIS
LIN {X -0.056,Y -673.225,Z 724.552,A 0.000,B 0.000,C 90.000,E1 315.445} C_DIS
LIN {X 0.032,Y -676.360,Z 724.547,A 0.000,B 0.000,C 90.000,E1 314.474} C_DIS
LIN {X -0.272,Y -680.004,Z 724.540,A 0.000,B 0.000,C 90.000,E1 313.299} C_DIS
LIN {X -0.059,Y -682.773,Z 724.535,A 0.000,B 0.000,C 90.000,E1 312.324} C_DIS
LIN {X 0.143,Y -685.338,Z 724.530,A 0.000,B 0.000,C 90.000,E1 311.353} C_DIS
LIN {X -0.014,Y -687.617,Z 724.525,A 0.000,B 0.000,C 90.000,E1 310.415} C_DIS
LIN {X -0.277,Y -689.270,Z 724.521,A 0.000,B 0.000,C 90.000,E1 309.725} C_DIS
LIN {X 0.066,Y -691.128,Z 724.515,A 0.000,B 0.000,C 90.000,E1 308.749} C_DIS
LIN {X -0.001,Y -692.734,Z 724.510,A 0.000,B 0.000,C 90.000,E1 307.810} C_DIS
LIN {X 0.012,Y -694.433,Z 724.504,A 0.000,B 0.000,C 90.000,E1 306.629} C_DIS
LIN {X 0.190,Y -695.879,Z 724.497,A 0.000,B 0.000,C 90.000,E1 305.438} C_DIS
LIN {X -0.232,Y -696.804,Z 724.492,A 0.000,B 0.000,C 90.000,E1 304.532} C_DIS
LIN {X -0.122,Y -698.257,Z 724.483,A 0.000,B 0.000,C 90.000,E1 302.880} C_DIS
LIN {X -0.018,Y -699.403,Z 724.475,A 0.000,B 0.000,C 90.000,E1 301.465} C_DIS
LIN {X 0.163,Y -699.932,Z 724.471,A 0.000,B 0.000,C 90.000,E1 300.747} C_DIS
LIN {X 0.103,Y -700.281,Z 724.467,A 0.000,B 0.000,C 90.000,E1 300.050} C_DIS
LIN {X 0.221,Y -700.617,Z 724.461,A 0.000,B 0.000,C 90.000,E1 298.871} C_DIS
LIN {X 0.016,Y -700.955,Z 724.454,A 0.000,B 0.000,C 90.000,E1 297.719} C_DIS
LIN {X 0.306,Y -701.828,Z 724.442,A 0.000,B 0.000,C 90.000,E1 295.591} C_DIS
LIN {X -0.075,Y -701.990,Z 724.440,A 0.000,B 0.000,C 90.000,E1 295.155} C_DIS
LIN {X -0.158,Y -701.821,Z 724.437,A 0.000,B 0.000,C 90.000,E1 294.695} C_DIS
LIN {X -0.174,Y -701.487,Z 724.436,A 0.000,B 0.000,C 90.000,E1 294.463} C_DIS
LIN {X 0.374,Y -699.917,Z 724.433,A 0.000,B 0.000,C 90.000,E1 293.951} C_DIS
LIN {X -0.279,Y -698.701,Z 724.432,A 0.000,B 0.000,C 90.000,E1 293.770} C_DIS
LIN {X -0.145,Y -697.617,Z 724.431,A 0.000,B 0.000,C 90.000,E1 293.643} C_DIS
LIN {X -0.174,Y -692.155,Z 724.429,A 0.000,B 0.000,C 90.000,E1 293.206} C_DIS
LIN {X 0.074,Y -690.251,Z 724.428,A 0.000,B 0.000,C 90.000,E1 293.078} C_DIS
LIN {X 0.176,Y -685.548,Z 724.427,A 0.000,B 0.000,C 90.000,E1 292.898} C_DIS
LIN {X 0.029,Y -677.044,Z 724.426,A 0.000,B 0.000,C 90.000,E1 292.695} C_DIS
LIN {X 0.185,Y -659.616,Z 724.425,A 0.000,B 0.000,C 90.000,E1 292.461} C_DIS
LIN {X -0.179,Y -646.031,Z 724.424,A 0.000,B 0.000,C 90.000,E1 292.280} C_DIS
LIN {X -0.036,Y -636.183,Z 724.423,A 0.000,B 0.000,C 90.000,E1 292.078} C_DIS
LIN {X -0.040,Y -622.728,Z 724.421,A 0.000,B 0.000,C 90.000,E1 291.770} C_DIS
LIN {X -0.190,Y -605.680,Z 724.418,A 0.000,B 0.000,C 90.000,E1 291.334} C_DIS
LIN {X 0.171,Y -577.533,Z 724.414,A 0.000,B 0.000,C 90.000,E1 290.482} C_DIS
LIN {X 0.071,Y -566.962,Z 724.412,A 0.000,B 0.000,C 90.000,E1 290.194} C_DIS
LIN {X 0.060,Y -561.136,Z 724.411,A 0.000,B 0.000,C 90.000,E1 289.993} C_DIS
LIN {X 0.019,Y -558.012,Z 724.410,A 0.000,B 0.000,C 90.000,E1 289.812} C_DIS
LIN {X 0.103,Y -556.462,Z 724.410,A 0.000,B 0.000,C 90.000,E1 289.704} C_DIS
LIN {X 0.073,Y -556.424,Z 724.410,A 0.000,B 0.000,C 90.000,E1 289.704} C_DIS
LIN {X -0.301,Y -555.503,Z 724.409,A 0.000,B 0.000,C 90.000,E1 289.577} C_DIS
LIN {X -0.280,Y -554.817,Z 724.406,A 0.000,B 0.000,C 90.000,E1 289.087} C_DIS
LIN {X 0.153,Y -554.463,Z 724.400,A 0.000,B 0.000,C 90.000,E1 288.000} C_DIS
LIN {X -0.162,Y -553.689,Z 724.389,A 0.000,B 0.000,C 90.000,E1 286.079} C_DIS
LIN {X -0.122,Y -553.005,Z 724.378,A 0.000,B 0.000,C 90.000,E1 284.120} C_DIS
LIN {X 0.300,Y -552.398,Z 724.368,A 0.000,B 0.000,C 90.000,E1 282.119} C_DIS
LIN {X -0.059,Y -551.589,Z 724.357,A 0.000,B 0.000,C 90.000,E1 280.197} C_DIS
LIN {X -0.117,Y -550.938,Z 724.349,A 0.000,B 0.000,C 90.000,E1 278.803} C_DIS
LIN {X -0.056,Y -550.009,Z 724.338,A 0.000,B 0.000,C 90.000,E1 276.834} C_DIS
LIN {X -0.143,Y -549.315,Z 724.327,A 0.000,B 0.000,C 90.000,E1 274.878} C_DIS
LIN {X 0.124,Y -548.940,Z 724.321,A 0.000,B 0.000,C 90.000,E1 273.726} C_DIS
LIN {X -0.106,Y -548.247,Z 724.311,A 0.000,B 0.000,C 90.000,E1 272.064} C_DIS
LIN {X 0.104,Y -547.763,Z 724.305,A 0.000,B 0.000,C 90.000,E1 270.917} C_DIS
LIN {X -0.208,Y -546.939,Z 724.297,A 0.000,B 0.000,C 90.000,E1 269.542} C_DIS
LIN {X 0.025,Y -546.082,Z 724.290,A 0.000,B 0.000,C 90.000,E1 268.108} C_DIS
LIN {X -0.263,Y -545.004,Z 724.280,A 0.000,B 0.000,C 90.000,E1 266.445} C_DIS
LIN {X -0.008,Y -543.798,Z 724.271,A 0.000,B 0.000,C 90.000,E1 264.723} C_DIS
LIN {X 0.250,Y -542.782,Z 724.263,A 0.000,B 0.000,C 90.000,E1 263.280} C_DIS
LIN {X -0.045,Y -541.591,Z 724.255,A 0.000,B 0.000,C 90.000,E1 261.894} C_DIS
LIN {X -0.209,Y -540.149,Z 724.246,A 0.000,B 0.000,C 90.000,E1 260.208} C_DIS
LIN {X -0.266,Y -538.191,Z 724.233,A 0.000,B 0.000,C 90.000,E1 257.937} C_DIS
LIN {X 0.177,Y -536.966,Z 724.225,A 0.000,B 0.000,C 90.000,E1 256.464} C_DIS
LIN {X 0.021,Y -535.915,Z 724.219,A 0.000,B 0.000,C 90.000,E1 255.338} C_DIS
LIN {X 0.132,Y -533.805,Z 724.207,A 0.000,B 0.000,C 90.000,E1 253.323} C_DIS
LIN {X -0.209,Y -532.061,Z 724.198,A 0.000,B 0.000,C 90.000,E1 251.638} C_DIS
LIN {X 0.195,Y -531.073,Z 724.193,A 0.000,B 0.000,C 90.000,E1 250.732} C_DIS
LIN {X -0.223,Y -529.144,Z 724.185,A 0.000,B 0.000,C 90.000,E1 249.337} C_DIS
LIN {X 0.016,Y -527.599,Z 724.179,A 0.000,B 0.000,C 90.000,E1 248.156} C_DIS
LIN {X -0.111,Y -525.054,Z 724.169,A 0.000,B 0.000,C 90.000,E1 246.433} C_DIS
LIN {X -0.037,Y -522.712,Z 724.161,A 0.000,B 0.000,C 90.000,E1 244.973} C_DIS
LIN {X -0.144,Y -520.823,Z 724.155,A 0.000,B 0.000,C 90.000,E1 243.819} C_DIS
LIN {X 0.049,Y -519.254,Z 724.150,A 0.000,B 0.000,C 90.000,E1 242.922} C_DIS
LIN {X -0.110,Y -517.010,Z 724.143,A 0.000,B 0.000,C 90.000,E1 241.769} C_DIS
LIN {X 0.043,Y -514.102,Z 724.135,A 0.000,B 0.000,C 90.000,E1 240.284} C_DIS
LIN {X 0.208,Y -511.118,Z 724.127,A 0.000,B 0.000,C 90.000,E1 238.791} C_DIS
LIN {X 0.054,Y -508.030,Z 724.119,A 0.000,B 0.000,C 90.000,E1 237.327} C_DIS
LIN {X -0.311,Y -504.887,Z 724.110,A 0.000,B 0.000,C 90.000,E1 235.881} C_DIS
LIN {X -0.220,Y -502.920,Z 724.105,A 0.000,B 0.000,C 90.000,E1 234.975} C_DIS
LIN {X 0.025,Y -500.046,Z 724.099,A 0.000,B 0.000,C 90.000,E1 233.749} C_DIS
LIN {X -0.069,Y -497.038,Z 724.092,A 0.000,B 0.000,C 90.000,E1 232.557} C_DIS
LIN {X 0.120,Y -490.989,Z 724.079,A 0.000,B 0.000,C 90.000,E1 230.114} C_DIS
LIN {X -0.070,Y -486.058,Z 724.067,A 0.000,B 0.000,C 90.000,E1 228.000} C_DIS
LIN {X -0.150,Y -483.243,Z 724.060,A 0.000,B 0.000,C 90.000,E1 226.782} C_DIS
LIN {X -0.166,Y -479.820,Z 724.051,A 0.000,B 0.000,C 90.000,E1 225.243} C_DIS
LIN {X -0.025,Y -475.173,Z 724.039,A 0.000,B 0.000,C 90.000,E1 223.056} C_DIS
LIN {X 0.265,Y -471.229,Z 724.029,A 0.000,B 0.000,C 90.000,E1 221.148} C_DIS
LIN {X -0.033,Y -468.527,Z 724.022,A 0.000,B 0.000,C 90.000,E1 219.930} C_DIS
LIN {X 0.112,Y -465.010,Z 724.013,A 0.000,B 0.000,C 90.000,E1 218.338} C_DIS
LIN {X -0.180,Y -458.836,Z 723.997,A 0.000,B 0.000,C 90.000,E1 215.518} C_DIS
LIN {X -0.191,Y -453.908,Z 723.983,A 0.000,B 0.000,C 90.000,E1 212.959} C_DIS
LIN {X 0.162,Y -449.145,Z 723.969,A 0.000,B 0.000,C 90.000,E1 210.335} C_DIS
LIN {X -0.071,Y -446.081,Z 723.960,A 0.000,B 0.000,C 90.000,E1 208.743} C_DIS
LIN {X -0.187,Y -443.131,Z 723.951,A 0.000,B 0.000,C 90.000,E1 207.129} C_DIS
LIN {X -0.002,Y -440.741,Z 723.943,A 0.000,B 0.000,C 90.000,E1 205.796} C_DIS
LIN {X -0.159,Y -436.523,Z 723.931,A 0.000,B 0.000,C 90.000,E1 203.515} C_DIS
LIN {X -0.030,Y -433.456,Z 723.921,A 0.000,B 0.000,C 90.000,E1 201.844} C_DIS
LIN {X 0.032,Y -430.368,Z 723.912,A 0.000,B 0.000,C 90.000,E1 200.174} C_DIS
LIN {X -0.057,Y -426.727,Z 723.901,A 0.000,B 0.000,C 90.000,E1 198.181} C_DIS
LIN {X -0.015,Y -423.521,Z 723.892,A 0.000,B 0.000,C 90.000,E1 196.496} C_DIS
LIN {X 0.125,Y -418.645,Z 723.877,A 0.000,B 0.000,C 90.000,E1 193.772} C_DIS
LIN {X -0.173,Y -415.003,Z 723.865,A 0.000,B 0.000,C 90.000,E1 191.771} C_DIS
LIN {X -0.176,Y -410.224,Z 723.850,A 0.000,B 0.000,C 90.000,E1 189.029} C_DIS
LIN {X -0.127,Y -406.387,Z 723.837,A 0.000,B 0.000,C 90.000,E1 186.606} C_DIS
LIN {X 0.183,Y -402.775,Z 723.823,A 0.000,B 0.000,C 90.000,E1 184.131} C_DIS
LIN {X -0.018,Y -399.923,Z 723.812,A 0.000,B 0.000,C 90.000,E1 182.064} C_DIS
